(* IEC 61131-3 sources: TIA2AX/tests/test_projects/expected/HW_2200330_V18/ST80_PLC, 6 files *)

(* ---- HwInputs.st ---- *)
TYPE
	HwInputs : STRUCT
		ST80_1_DM260_EB_Box_Acquisition_Status_1 AT %B1205 : ARRAY[0..2] OF BYTE;
		ST80_1_DM260_EB_Box_Results_Status_1 AT %B1208 : BYTE;
		ST80_1_DM260_EB_Box_Soft_Event_Control_1 AT %B1209 : BYTE;
		ST80_1_DM260_EB_Box_Result_Data_64_bytes_1 AT %B1382 : ARRAY[0..71] OF BYTE;
		ST80_1_DM260_PB_Box_Acquisition_Status_1 AT %B1200 : ARRAY[0..2] OF BYTE;
		ST80_1_DM260_PB_Box_Results_Status_1 AT %B1203 : BYTE;
		ST80_1_DM260_PB_Box_Soft_Event_Control_1 AT %B1204 : BYTE;
		ST80_1_DM260_PB_Box_Result_Data_64_bytes_1 AT %B1210 : ARRAY[0..71] OF BYTE;
		ST80_ET200SP_2_11M1 AT %B600 : DWORD;
		ST80_ET200SP_2_11M2 AT %B604 : DWORD;
		ST80_ET200SP_2_11M3 AT %B608 : DWORD;
		ST80_ET200SP_2_11M4 AT %B612 : DWORD;
		ST80_ET200SP_2_12M1 AT %B616 : DWORD;
		ST80_ET200SP_2_12M2 AT %B620 : DWORD;
		ST80_ET200SP_2_12M3 AT %B624 : DWORD;
		ST80_ET200SP_2_12M4 AT %B628 : DWORD;
		ST80_ET200SP_2_13M1 AT %B632 : DWORD;
		ST80_ET200SP_2_13M2 AT %B636 : DWORD;
		ST80_ET200SP_2_13M3 AT %B640 : DWORD;
		ST80_ET200SP_2_13M4 AT %B644 : DWORD;
		ST80_1_TZ535_PN_In_Out_32_byte_1 AT %B1800 : ARRAY[0..31] OF BYTE;
		ST80_1_DM260_Housing_Acquisition_Status_1 AT %B1000 : ARRAY[0..2] OF BYTE;
		ST80_1_DM260_Housing_Results_Status_1 AT %B1003 : BYTE;
		ST80_1_DM260_Housing_Soft_Event_Control_1 AT %B1004 : BYTE;
		ST80_1_DM260_Housing_Result_Data_64_bytes_1 AT %B1010 : ARRAY[0..71] OF BYTE;
		ST80_ET200SP_CM_4xIO_Link_1 AT %B100 : ARRAY[0..31] OF BYTE;
		ST80_ET200SP_CM_4xIO_Link_2 AT %B132 : ARRAY[0..31] OF BYTE;
		ST80_ET200SP_CM_4xIO_Link_3 AT %B164 : ARRAY[0..31] OF BYTE;
		ST80_ET200SP_DI_16x24VDC_ST_1 AT %B0 : WORD;
		ST80_ET200SP_DI_16x24VDC_ST_2 AT %B2 : WORD;
		ST80_ET200SP_DI_16x24VDC_ST_3 AT %B4 : WORD;
		ST80_ET200SP_DI_16x24VDC_ST_4 AT %B6 : WORD;
	END_STRUCT;
END_TYPE

(* ---- HwOutputs.st ---- *)
TYPE
	HwOutputs : STRUCT
		ST80_1_DM260_EB_Box_Acquisition_Control_1 AT %B1201 : BYTE;
		ST80_1_DM260_EB_Box_Results_Control_1 AT %B1205 : BYTE;
		ST80_1_DM260_EB_Box_Soft_Event_Control_1 AT %B1206 : BYTE;
		ST80_1_DM260_EB_Box_User_Data_64_bytes_1 AT %B1378 : ARRAY[0..67] OF BYTE;
		ST80_1_DM260_PB_Box_Acquisition_Control_1 AT %B1200 : BYTE;
		ST80_1_DM260_PB_Box_Results_Control_1 AT %B1203 : BYTE;
		ST80_1_DM260_PB_Box_Soft_Event_Control_1 AT %B1204 : BYTE;
		ST80_1_DM260_PB_Box_User_Data_64_bytes_1 AT %B1210 : ARRAY[0..67] OF BYTE;
		ST80_ET200SP_2_11M1 AT %B600 : WORD;
		ST80_ET200SP_2_11M2 AT %B604 : WORD;
		ST80_ET200SP_2_11M3 AT %B608 : WORD;
		ST80_ET200SP_2_11M4 AT %B612 : WORD;
		ST80_ET200SP_2_12M1 AT %B616 : WORD;
		ST80_ET200SP_2_12M2 AT %B620 : WORD;
		ST80_ET200SP_2_12M3 AT %B624 : WORD;
		ST80_ET200SP_2_12M4 AT %B628 : WORD;
		ST80_ET200SP_2_13M1 AT %B632 : WORD;
		ST80_ET200SP_2_13M2 AT %B636 : WORD;
		ST80_ET200SP_2_13M3 AT %B640 : WORD;
		ST80_ET200SP_2_13M4 AT %B644 : WORD;
		ST80_1_TZ535_PN_In_Out_32_byte_1 AT %B1800 : ARRAY[0..31] OF BYTE;
		ST80_1_DM260_Housing_Acquisition_Control_1 AT %B1000 : BYTE;
		ST80_1_DM260_Housing_Results_Control_1 AT %B1003 : BYTE;
		ST80_1_DM260_Housing_Soft_Event_Control_1 AT %B1004 : BYTE;
		ST80_1_DM260_Housing_User_Data_64_bytes_1 AT %B1010 : ARRAY[0..67] OF BYTE;
		ST80_CPX_MPA1S_VMPA1_FB_EMS_8_8DO_1 AT %B200 : BYTE;
		ST80_CPX_MPA1S_VMPA1_FB_EMS_8_8DO_2 AT %B201 : BYTE;
		ST80_CPX_MPA2S_VMPA2_FB_EMS_4_4DO_1 AT %B202 : BYTE;
		ST80_CPX_MPA1S_VMPA1_FB_EMS_8_8DO_3 AT %B203 : BYTE;
		ST80_CPX_MPA2S_VMPA2_FB_EMS_4_4DO_2 AT %B204 : BYTE;
		ST80_CPX_MPA1S_VMPA1_FB_EMS_8_8DO_4 AT %B205 : BYTE;
		ST80_CPX_MPA1S_VMPA1_FB_EMS_8_8DO_5 AT %B206 : BYTE;
		ST80_CPX_MPA1G_VMPA1_FB_EMG_8_8DO_1 AT %B207 : BYTE;
		ST80_CPX_MPA1G_VMPA1_FB_EMG_8_8DO_2 AT %B208 : BYTE;
		ST80_CPX_MPA2G_VMPA2_FB_EMG_4_4DO_1 AT %B209 : BYTE;
		ST80_CPX_MPA1G_VMPA1_FB_EMG_8_8DO_3 AT %B210 : BYTE;
		ST80_CPX_MPA1G_VMPA1_FB_EMG_8_8DO_4 AT %B211 : BYTE;
		ST80_CPX_MPA1G_VMPA1_FB_EMG_8_8DO_5 AT %B212 : BYTE;
		ST80_CPX_MPA1G_VMPA1_FB_EMG_8_8DO_6 AT %B213 : BYTE;
		ST80_ET200SP_CM_4xIO_Link_1 AT %B100 : ARRAY[0..31] OF BYTE;
		ST80_ET200SP_CM_4xIO_Link_2 AT %B132 : ARRAY[0..31] OF BYTE;
		ST80_ET200SP_CM_4xIO_Link_3 AT %B164 : ARRAY[0..31] OF BYTE;
		ST80_ET200SP_DQ_16x24VDC_0_5A_ST_1 AT %B0 : WORD;
		ST80_ET200SP_DQ_16x24VDC_0_5A_ST_2 AT %B2 : WORD;
		ST80_ET200SP_DQ_16x24VDC_0_5A_ST_3 AT %B4 : WORD;
	END_STRUCT;
END_TYPE

(* ---- PlcInputs.st ---- *)
TYPE
	PlcInputs : STRUCT
		ST80_1_DM260_EB_Box_Acquisition_Status_1 : ARRAY[0..2] OF BYTE;
		ST80_1_DM260_EB_Box_Results_Status_1 : BYTE;
		ST80_1_DM260_EB_Box_Soft_Event_Control_1 : BYTE;
		ST80_1_DM260_EB_Box_Result_Data_64_bytes_1 : ARRAY[0..71] OF BYTE;
		ST80_1_DM260_PB_Box_Acquisition_Status_1 : ARRAY[0..2] OF BYTE;
		ST80_1_DM260_PB_Box_Results_Status_1 : BYTE;
		ST80_1_DM260_PB_Box_Soft_Event_Control_1 : BYTE;
		ST80_1_DM260_PB_Box_Result_Data_64_bytes_1 : ARRAY[0..71] OF BYTE;
		ST80_ET200SP_2_11M1 : DWORD;
		ST80_ET200SP_2_11M2 : DWORD;
		ST80_ET200SP_2_11M3 : DWORD;
		ST80_ET200SP_2_11M4 : DWORD;
		ST80_ET200SP_2_12M1 : DWORD;
		ST80_ET200SP_2_12M2 : DWORD;
		ST80_ET200SP_2_12M3 : DWORD;
		ST80_ET200SP_2_12M4 : DWORD;
		ST80_ET200SP_2_13M1 : DWORD;
		ST80_ET200SP_2_13M2 : DWORD;
		ST80_ET200SP_2_13M3 : DWORD;
		ST80_ET200SP_2_13M4 : DWORD;
		ST80_1_TZ535_PN_In_Out_32_byte_1 : ARRAY[0..31] OF BYTE;
		ST80_1_DM260_Housing_Acquisition_Status_1 : ARRAY[0..2] OF BYTE;
		ST80_1_DM260_Housing_Results_Status_1 : BYTE;
		ST80_1_DM260_Housing_Soft_Event_Control_1 : BYTE;
		ST80_1_DM260_Housing_Result_Data_64_bytes_1 : ARRAY[0..71] OF BYTE;
		ST80_ET200SP_CM_4xIO_Link_1 : ARRAY[0..31] OF BYTE;
		ST80_ET200SP_CM_4xIO_Link_2 : ARRAY[0..31] OF BYTE;
		ST80_ET200SP_CM_4xIO_Link_3 : ARRAY[0..31] OF BYTE;
		ST80_ET200SP_DI_16x24VDC_ST_1 : WORD;
		ST80_ET200SP_DI_16x24VDC_ST_2 : WORD;
		ST80_ET200SP_DI_16x24VDC_ST_3 : WORD;
		ST80_ET200SP_DI_16x24VDC_ST_4 : WORD;
	END_STRUCT;
END_TYPE

(* ---- PlcOutputs.st ---- *)
TYPE
	PlcOutputs : STRUCT
		ST80_1_DM260_EB_Box_Acquisition_Control_1 : BYTE;
		ST80_1_DM260_EB_Box_Results_Control_1 : BYTE;
		ST80_1_DM260_EB_Box_Soft_Event_Control_1 : BYTE;
		ST80_1_DM260_EB_Box_User_Data_64_bytes_1 : ARRAY[0..67] OF BYTE;
		ST80_1_DM260_PB_Box_Acquisition_Control_1 : BYTE;
		ST80_1_DM260_PB_Box_Results_Control_1 : BYTE;
		ST80_1_DM260_PB_Box_Soft_Event_Control_1 : BYTE;
		ST80_1_DM260_PB_Box_User_Data_64_bytes_1 : ARRAY[0..67] OF BYTE;
		ST80_ET200SP_2_11M1 : WORD;
		ST80_ET200SP_2_11M2 : WORD;
		ST80_ET200SP_2_11M3 : WORD;
		ST80_ET200SP_2_11M4 : WORD;
		ST80_ET200SP_2_12M1 : WORD;
		ST80_ET200SP_2_12M2 : WORD;
		ST80_ET200SP_2_12M3 : WORD;
		ST80_ET200SP_2_12M4 : WORD;
		ST80_ET200SP_2_13M1 : WORD;
		ST80_ET200SP_2_13M2 : WORD;
		ST80_ET200SP_2_13M3 : WORD;
		ST80_ET200SP_2_13M4 : WORD;
		ST80_1_TZ535_PN_In_Out_32_byte_1 : ARRAY[0..31] OF BYTE;
		ST80_1_DM260_Housing_Acquisition_Control_1 : BYTE;
		ST80_1_DM260_Housing_Results_Control_1 : BYTE;
		ST80_1_DM260_Housing_Soft_Event_Control_1 : BYTE;
		ST80_1_DM260_Housing_User_Data_64_bytes_1 : ARRAY[0..67] OF BYTE;
		ST80_CPX_MPA1S_VMPA1_FB_EMS_8_8DO_1 : BYTE;
		ST80_CPX_MPA1S_VMPA1_FB_EMS_8_8DO_2 : BYTE;
		ST80_CPX_MPA2S_VMPA2_FB_EMS_4_4DO_1 : BYTE;
		ST80_CPX_MPA1S_VMPA1_FB_EMS_8_8DO_3 : BYTE;
		ST80_CPX_MPA2S_VMPA2_FB_EMS_4_4DO_2 : BYTE;
		ST80_CPX_MPA1S_VMPA1_FB_EMS_8_8DO_4 : BYTE;
		ST80_CPX_MPA1S_VMPA1_FB_EMS_8_8DO_5 : BYTE;
		ST80_CPX_MPA1G_VMPA1_FB_EMG_8_8DO_1 : BYTE;
		ST80_CPX_MPA1G_VMPA1_FB_EMG_8_8DO_2 : BYTE;
		ST80_CPX_MPA2G_VMPA2_FB_EMG_4_4DO_1 : BYTE;
		ST80_CPX_MPA1G_VMPA1_FB_EMG_8_8DO_3 : BYTE;
		ST80_CPX_MPA1G_VMPA1_FB_EMG_8_8DO_4 : BYTE;
		ST80_CPX_MPA1G_VMPA1_FB_EMG_8_8DO_5 : BYTE;
		ST80_CPX_MPA1G_VMPA1_FB_EMG_8_8DO_6 : BYTE;
		ST80_ET200SP_CM_4xIO_Link_1 : ARRAY[0..31] OF BYTE;
		ST80_ET200SP_CM_4xIO_Link_2 : ARRAY[0..31] OF BYTE;
		ST80_ET200SP_CM_4xIO_Link_3 : ARRAY[0..31] OF BYTE;
		ST80_ET200SP_DQ_16x24VDC_0_5A_ST_1 : WORD;
		ST80_ET200SP_DQ_16x24VDC_0_5A_ST_2 : WORD;
		ST80_ET200SP_DQ_16x24VDC_0_5A_ST_3 : WORD;
	END_STRUCT;
END_TYPE

(* ---- CopyInputs.st ---- *)
FUNCTION CopyInputs
	VAR_EXTERNAL
		HwInputs : HwInputs;
		PlcInputs : PlcInputs;
	END_VAR
	PlcInputs.ST80_1_DM260_EB_Box_Acquisition_Status_1[0] := HwInputs.ST80_1_DM260_EB_Box_Acquisition_Status_1[0];
	PlcInputs.ST80_1_DM260_EB_Box_Acquisition_Status_1[1] := HwInputs.ST80_1_DM260_EB_Box_Acquisition_Status_1[1];
	PlcInputs.ST80_1_DM260_EB_Box_Acquisition_Status_1[2] := HwInputs.ST80_1_DM260_EB_Box_Acquisition_Status_1[2];
	PlcInputs.ST80_1_DM260_EB_Box_Results_Status_1 := HwInputs.ST80_1_DM260_EB_Box_Results_Status_1;
	PlcInputs.ST80_1_DM260_EB_Box_Soft_Event_Control_1 := HwInputs.ST80_1_DM260_EB_Box_Soft_Event_Control_1;
	PlcInputs.ST80_1_DM260_EB_Box_Result_Data_64_bytes_1[0] := HwInputs.ST80_1_DM260_EB_Box_Result_Data_64_bytes_1[0];
	PlcInputs.ST80_1_DM260_EB_Box_Result_Data_64_bytes_1[1] := HwInputs.ST80_1_DM260_EB_Box_Result_Data_64_bytes_1[1];
	PlcInputs.ST80_1_DM260_EB_Box_Result_Data_64_bytes_1[2] := HwInputs.ST80_1_DM260_EB_Box_Result_Data_64_bytes_1[2];
	PlcInputs.ST80_1_DM260_EB_Box_Result_Data_64_bytes_1[3] := HwInputs.ST80_1_DM260_EB_Box_Result_Data_64_bytes_1[3];
	PlcInputs.ST80_1_DM260_EB_Box_Result_Data_64_bytes_1[4] := HwInputs.ST80_1_DM260_EB_Box_Result_Data_64_bytes_1[4];
	PlcInputs.ST80_1_DM260_EB_Box_Result_Data_64_bytes_1[5] := HwInputs.ST80_1_DM260_EB_Box_Result_Data_64_bytes_1[5];
	PlcInputs.ST80_1_DM260_EB_Box_Result_Data_64_bytes_1[6] := HwInputs.ST80_1_DM260_EB_Box_Result_Data_64_bytes_1[6];
	PlcInputs.ST80_1_DM260_EB_Box_Result_Data_64_bytes_1[7] := HwInputs.ST80_1_DM260_EB_Box_Result_Data_64_bytes_1[7];
	PlcInputs.ST80_1_DM260_EB_Box_Result_Data_64_bytes_1[8] := HwInputs.ST80_1_DM260_EB_Box_Result_Data_64_bytes_1[8];
	PlcInputs.ST80_1_DM260_EB_Box_Result_Data_64_bytes_1[9] := HwInputs.ST80_1_DM260_EB_Box_Result_Data_64_bytes_1[9];
	PlcInputs.ST80_1_DM260_EB_Box_Result_Data_64_bytes_1[10] := HwInputs.ST80_1_DM260_EB_Box_Result_Data_64_bytes_1[10];
	PlcInputs.ST80_1_DM260_EB_Box_Result_Data_64_bytes_1[11] := HwInputs.ST80_1_DM260_EB_Box_Result_Data_64_bytes_1[11];
	PlcInputs.ST80_1_DM260_EB_Box_Result_Data_64_bytes_1[12] := HwInputs.ST80_1_DM260_EB_Box_Result_Data_64_bytes_1[12];
	PlcInputs.ST80_1_DM260_EB_Box_Result_Data_64_bytes_1[13] := HwInputs.ST80_1_DM260_EB_Box_Result_Data_64_bytes_1[13];
	PlcInputs.ST80_1_DM260_EB_Box_Result_Data_64_bytes_1[14] := HwInputs.ST80_1_DM260_EB_Box_Result_Data_64_bytes_1[14];
	PlcInputs.ST80_1_DM260_EB_Box_Result_Data_64_bytes_1[15] := HwInputs.ST80_1_DM260_EB_Box_Result_Data_64_bytes_1[15];
	PlcInputs.ST80_1_DM260_EB_Box_Result_Data_64_bytes_1[16] := HwInputs.ST80_1_DM260_EB_Box_Result_Data_64_bytes_1[16];
	PlcInputs.ST80_1_DM260_EB_Box_Result_Data_64_bytes_1[17] := HwInputs.ST80_1_DM260_EB_Box_Result_Data_64_bytes_1[17];
	PlcInputs.ST80_1_DM260_EB_Box_Result_Data_64_bytes_1[18] := HwInputs.ST80_1_DM260_EB_Box_Result_Data_64_bytes_1[18];
	PlcInputs.ST80_1_DM260_EB_Box_Result_Data_64_bytes_1[19] := HwInputs.ST80_1_DM260_EB_Box_Result_Data_64_bytes_1[19];
	PlcInputs.ST80_1_DM260_EB_Box_Result_Data_64_bytes_1[20] := HwInputs.ST80_1_DM260_EB_Box_Result_Data_64_bytes_1[20];
	PlcInputs.ST80_1_DM260_EB_Box_Result_Data_64_bytes_1[21] := HwInputs.ST80_1_DM260_EB_Box_Result_Data_64_bytes_1[21];
	PlcInputs.ST80_1_DM260_EB_Box_Result_Data_64_bytes_1[22] := HwInputs.ST80_1_DM260_EB_Box_Result_Data_64_bytes_1[22];
	PlcInputs.ST80_1_DM260_EB_Box_Result_Data_64_bytes_1[23] := HwInputs.ST80_1_DM260_EB_Box_Result_Data_64_bytes_1[23];
	PlcInputs.ST80_1_DM260_EB_Box_Result_Data_64_bytes_1[24] := HwInputs.ST80_1_DM260_EB_Box_Result_Data_64_bytes_1[24];
	PlcInputs.ST80_1_DM260_EB_Box_Result_Data_64_bytes_1[25] := HwInputs.ST80_1_DM260_EB_Box_Result_Data_64_bytes_1[25];
	PlcInputs.ST80_1_DM260_EB_Box_Result_Data_64_bytes_1[26] := HwInputs.ST80_1_DM260_EB_Box_Result_Data_64_bytes_1[26];
	PlcInputs.ST80_1_DM260_EB_Box_Result_Data_64_bytes_1[27] := HwInputs.ST80_1_DM260_EB_Box_Result_Data_64_bytes_1[27];
	PlcInputs.ST80_1_DM260_EB_Box_Result_Data_64_bytes_1[28] := HwInputs.ST80_1_DM260_EB_Box_Result_Data_64_bytes_1[28];
	PlcInputs.ST80_1_DM260_EB_Box_Result_Data_64_bytes_1[29] := HwInputs.ST80_1_DM260_EB_Box_Result_Data_64_bytes_1[29];
	PlcInputs.ST80_1_DM260_EB_Box_Result_Data_64_bytes_1[30] := HwInputs.ST80_1_DM260_EB_Box_Result_Data_64_bytes_1[30];
	PlcInputs.ST80_1_DM260_EB_Box_Result_Data_64_bytes_1[31] := HwInputs.ST80_1_DM260_EB_Box_Result_Data_64_bytes_1[31];
	PlcInputs.ST80_1_DM260_EB_Box_Result_Data_64_bytes_1[32] := HwInputs.ST80_1_DM260_EB_Box_Result_Data_64_bytes_1[32];
	PlcInputs.ST80_1_DM260_EB_Box_Result_Data_64_bytes_1[33] := HwInputs.ST80_1_DM260_EB_Box_Result_Data_64_bytes_1[33];
	PlcInputs.ST80_1_DM260_EB_Box_Result_Data_64_bytes_1[34] := HwInputs.ST80_1_DM260_EB_Box_Result_Data_64_bytes_1[34];
	PlcInputs.ST80_1_DM260_EB_Box_Result_Data_64_bytes_1[35] := HwInputs.ST80_1_DM260_EB_Box_Result_Data_64_bytes_1[35];
	PlcInputs.ST80_1_DM260_EB_Box_Result_Data_64_bytes_1[36] := HwInputs.ST80_1_DM260_EB_Box_Result_Data_64_bytes_1[36];
	PlcInputs.ST80_1_DM260_EB_Box_Result_Data_64_bytes_1[37] := HwInputs.ST80_1_DM260_EB_Box_Result_Data_64_bytes_1[37];
	PlcInputs.ST80_1_DM260_EB_Box_Result_Data_64_bytes_1[38] := HwInputs.ST80_1_DM260_EB_Box_Result_Data_64_bytes_1[38];
	PlcInputs.ST80_1_DM260_EB_Box_Result_Data_64_bytes_1[39] := HwInputs.ST80_1_DM260_EB_Box_Result_Data_64_bytes_1[39];
	PlcInputs.ST80_1_DM260_EB_Box_Result_Data_64_bytes_1[40] := HwInputs.ST80_1_DM260_EB_Box_Result_Data_64_bytes_1[40];
	PlcInputs.ST80_1_DM260_EB_Box_Result_Data_64_bytes_1[41] := HwInputs.ST80_1_DM260_EB_Box_Result_Data_64_bytes_1[41];
	PlcInputs.ST80_1_DM260_EB_Box_Result_Data_64_bytes_1[42] := HwInputs.ST80_1_DM260_EB_Box_Result_Data_64_bytes_1[42];
	PlcInputs.ST80_1_DM260_EB_Box_Result_Data_64_bytes_1[43] := HwInputs.ST80_1_DM260_EB_Box_Result_Data_64_bytes_1[43];
	PlcInputs.ST80_1_DM260_EB_Box_Result_Data_64_bytes_1[44] := HwInputs.ST80_1_DM260_EB_Box_Result_Data_64_bytes_1[44];
	PlcInputs.ST80_1_DM260_EB_Box_Result_Data_64_bytes_1[45] := HwInputs.ST80_1_DM260_EB_Box_Result_Data_64_bytes_1[45];
	PlcInputs.ST80_1_DM260_EB_Box_Result_Data_64_bytes_1[46] := HwInputs.ST80_1_DM260_EB_Box_Result_Data_64_bytes_1[46];
	PlcInputs.ST80_1_DM260_EB_Box_Result_Data_64_bytes_1[47] := HwInputs.ST80_1_DM260_EB_Box_Result_Data_64_bytes_1[47];
	PlcInputs.ST80_1_DM260_EB_Box_Result_Data_64_bytes_1[48] := HwInputs.ST80_1_DM260_EB_Box_Result_Data_64_bytes_1[48];
	PlcInputs.ST80_1_DM260_EB_Box_Result_Data_64_bytes_1[49] := HwInputs.ST80_1_DM260_EB_Box_Result_Data_64_bytes_1[49];
	PlcInputs.ST80_1_DM260_EB_Box_Result_Data_64_bytes_1[50] := HwInputs.ST80_1_DM260_EB_Box_Result_Data_64_bytes_1[50];
	PlcInputs.ST80_1_DM260_EB_Box_Result_Data_64_bytes_1[51] := HwInputs.ST80_1_DM260_EB_Box_Result_Data_64_bytes_1[51];
	PlcInputs.ST80_1_DM260_EB_Box_Result_Data_64_bytes_1[52] := HwInputs.ST80_1_DM260_EB_Box_Result_Data_64_bytes_1[52];
	PlcInputs.ST80_1_DM260_EB_Box_Result_Data_64_bytes_1[53] := HwInputs.ST80_1_DM260_EB_Box_Result_Data_64_bytes_1[53];
	PlcInputs.ST80_1_DM260_EB_Box_Result_Data_64_bytes_1[54] := HwInputs.ST80_1_DM260_EB_Box_Result_Data_64_bytes_1[54];
	PlcInputs.ST80_1_DM260_EB_Box_Result_Data_64_bytes_1[55] := HwInputs.ST80_1_DM260_EB_Box_Result_Data_64_bytes_1[55];
	PlcInputs.ST80_1_DM260_EB_Box_Result_Data_64_bytes_1[56] := HwInputs.ST80_1_DM260_EB_Box_Result_Data_64_bytes_1[56];
	PlcInputs.ST80_1_DM260_EB_Box_Result_Data_64_bytes_1[57] := HwInputs.ST80_1_DM260_EB_Box_Result_Data_64_bytes_1[57];
	PlcInputs.ST80_1_DM260_EB_Box_Result_Data_64_bytes_1[58] := HwInputs.ST80_1_DM260_EB_Box_Result_Data_64_bytes_1[58];
	PlcInputs.ST80_1_DM260_EB_Box_Result_Data_64_bytes_1[59] := HwInputs.ST80_1_DM260_EB_Box_Result_Data_64_bytes_1[59];
	PlcInputs.ST80_1_DM260_EB_Box_Result_Data_64_bytes_1[60] := HwInputs.ST80_1_DM260_EB_Box_Result_Data_64_bytes_1[60];
	PlcInputs.ST80_1_DM260_EB_Box_Result_Data_64_bytes_1[61] := HwInputs.ST80_1_DM260_EB_Box_Result_Data_64_bytes_1[61];
	PlcInputs.ST80_1_DM260_EB_Box_Result_Data_64_bytes_1[62] := HwInputs.ST80_1_DM260_EB_Box_Result_Data_64_bytes_1[62];
	PlcInputs.ST80_1_DM260_EB_Box_Result_Data_64_bytes_1[63] := HwInputs.ST80_1_DM260_EB_Box_Result_Data_64_bytes_1[63];
	PlcInputs.ST80_1_DM260_EB_Box_Result_Data_64_bytes_1[64] := HwInputs.ST80_1_DM260_EB_Box_Result_Data_64_bytes_1[64];
	PlcInputs.ST80_1_DM260_EB_Box_Result_Data_64_bytes_1[65] := HwInputs.ST80_1_DM260_EB_Box_Result_Data_64_bytes_1[65];
	PlcInputs.ST80_1_DM260_EB_Box_Result_Data_64_bytes_1[66] := HwInputs.ST80_1_DM260_EB_Box_Result_Data_64_bytes_1[66];
	PlcInputs.ST80_1_DM260_EB_Box_Result_Data_64_bytes_1[67] := HwInputs.ST80_1_DM260_EB_Box_Result_Data_64_bytes_1[67];
	PlcInputs.ST80_1_DM260_EB_Box_Result_Data_64_bytes_1[68] := HwInputs.ST80_1_DM260_EB_Box_Result_Data_64_bytes_1[68];
	PlcInputs.ST80_1_DM260_EB_Box_Result_Data_64_bytes_1[69] := HwInputs.ST80_1_DM260_EB_Box_Result_Data_64_bytes_1[69];
	PlcInputs.ST80_1_DM260_EB_Box_Result_Data_64_bytes_1[70] := HwInputs.ST80_1_DM260_EB_Box_Result_Data_64_bytes_1[70];
	PlcInputs.ST80_1_DM260_EB_Box_Result_Data_64_bytes_1[71] := HwInputs.ST80_1_DM260_EB_Box_Result_Data_64_bytes_1[71];
	PlcInputs.ST80_1_DM260_PB_Box_Acquisition_Status_1[0] := HwInputs.ST80_1_DM260_PB_Box_Acquisition_Status_1[0];
	PlcInputs.ST80_1_DM260_PB_Box_Acquisition_Status_1[1] := HwInputs.ST80_1_DM260_PB_Box_Acquisition_Status_1[1];
	PlcInputs.ST80_1_DM260_PB_Box_Acquisition_Status_1[2] := HwInputs.ST80_1_DM260_PB_Box_Acquisition_Status_1[2];
	PlcInputs.ST80_1_DM260_PB_Box_Results_Status_1 := HwInputs.ST80_1_DM260_PB_Box_Results_Status_1;
	PlcInputs.ST80_1_DM260_PB_Box_Soft_Event_Control_1 := HwInputs.ST80_1_DM260_PB_Box_Soft_Event_Control_1;
	PlcInputs.ST80_1_DM260_PB_Box_Result_Data_64_bytes_1[0] := HwInputs.ST80_1_DM260_PB_Box_Result_Data_64_bytes_1[0];
	PlcInputs.ST80_1_DM260_PB_Box_Result_Data_64_bytes_1[1] := HwInputs.ST80_1_DM260_PB_Box_Result_Data_64_bytes_1[1];
	PlcInputs.ST80_1_DM260_PB_Box_Result_Data_64_bytes_1[2] := HwInputs.ST80_1_DM260_PB_Box_Result_Data_64_bytes_1[2];
	PlcInputs.ST80_1_DM260_PB_Box_Result_Data_64_bytes_1[3] := HwInputs.ST80_1_DM260_PB_Box_Result_Data_64_bytes_1[3];
	PlcInputs.ST80_1_DM260_PB_Box_Result_Data_64_bytes_1[4] := HwInputs.ST80_1_DM260_PB_Box_Result_Data_64_bytes_1[4];
	PlcInputs.ST80_1_DM260_PB_Box_Result_Data_64_bytes_1[5] := HwInputs.ST80_1_DM260_PB_Box_Result_Data_64_bytes_1[5];
	PlcInputs.ST80_1_DM260_PB_Box_Result_Data_64_bytes_1[6] := HwInputs.ST80_1_DM260_PB_Box_Result_Data_64_bytes_1[6];
	PlcInputs.ST80_1_DM260_PB_Box_Result_Data_64_bytes_1[7] := HwInputs.ST80_1_DM260_PB_Box_Result_Data_64_bytes_1[7];
	PlcInputs.ST80_1_DM260_PB_Box_Result_Data_64_bytes_1[8] := HwInputs.ST80_1_DM260_PB_Box_Result_Data_64_bytes_1[8];
	PlcInputs.ST80_1_DM260_PB_Box_Result_Data_64_bytes_1[9] := HwInputs.ST80_1_DM260_PB_Box_Result_Data_64_bytes_1[9];
	PlcInputs.ST80_1_DM260_PB_Box_Result_Data_64_bytes_1[10] := HwInputs.ST80_1_DM260_PB_Box_Result_Data_64_bytes_1[10];
	PlcInputs.ST80_1_DM260_PB_Box_Result_Data_64_bytes_1[11] := HwInputs.ST80_1_DM260_PB_Box_Result_Data_64_bytes_1[11];
	PlcInputs.ST80_1_DM260_PB_Box_Result_Data_64_bytes_1[12] := HwInputs.ST80_1_DM260_PB_Box_Result_Data_64_bytes_1[12];
	PlcInputs.ST80_1_DM260_PB_Box_Result_Data_64_bytes_1[13] := HwInputs.ST80_1_DM260_PB_Box_Result_Data_64_bytes_1[13];
	PlcInputs.ST80_1_DM260_PB_Box_Result_Data_64_bytes_1[14] := HwInputs.ST80_1_DM260_PB_Box_Result_Data_64_bytes_1[14];
	PlcInputs.ST80_1_DM260_PB_Box_Result_Data_64_bytes_1[15] := HwInputs.ST80_1_DM260_PB_Box_Result_Data_64_bytes_1[15];
	PlcInputs.ST80_1_DM260_PB_Box_Result_Data_64_bytes_1[16] := HwInputs.ST80_1_DM260_PB_Box_Result_Data_64_bytes_1[16];
	PlcInputs.ST80_1_DM260_PB_Box_Result_Data_64_bytes_1[17] := HwInputs.ST80_1_DM260_PB_Box_Result_Data_64_bytes_1[17];
	PlcInputs.ST80_1_DM260_PB_Box_Result_Data_64_bytes_1[18] := HwInputs.ST80_1_DM260_PB_Box_Result_Data_64_bytes_1[18];
	PlcInputs.ST80_1_DM260_PB_Box_Result_Data_64_bytes_1[19] := HwInputs.ST80_1_DM260_PB_Box_Result_Data_64_bytes_1[19];
	PlcInputs.ST80_1_DM260_PB_Box_Result_Data_64_bytes_1[20] := HwInputs.ST80_1_DM260_PB_Box_Result_Data_64_bytes_1[20];
	PlcInputs.ST80_1_DM260_PB_Box_Result_Data_64_bytes_1[21] := HwInputs.ST80_1_DM260_PB_Box_Result_Data_64_bytes_1[21];
	PlcInputs.ST80_1_DM260_PB_Box_Result_Data_64_bytes_1[22] := HwInputs.ST80_1_DM260_PB_Box_Result_Data_64_bytes_1[22];
	PlcInputs.ST80_1_DM260_PB_Box_Result_Data_64_bytes_1[23] := HwInputs.ST80_1_DM260_PB_Box_Result_Data_64_bytes_1[23];
	PlcInputs.ST80_1_DM260_PB_Box_Result_Data_64_bytes_1[24] := HwInputs.ST80_1_DM260_PB_Box_Result_Data_64_bytes_1[24];
	PlcInputs.ST80_1_DM260_PB_Box_Result_Data_64_bytes_1[25] := HwInputs.ST80_1_DM260_PB_Box_Result_Data_64_bytes_1[25];
	PlcInputs.ST80_1_DM260_PB_Box_Result_Data_64_bytes_1[26] := HwInputs.ST80_1_DM260_PB_Box_Result_Data_64_bytes_1[26];
	PlcInputs.ST80_1_DM260_PB_Box_Result_Data_64_bytes_1[27] := HwInputs.ST80_1_DM260_PB_Box_Result_Data_64_bytes_1[27];
	PlcInputs.ST80_1_DM260_PB_Box_Result_Data_64_bytes_1[28] := HwInputs.ST80_1_DM260_PB_Box_Result_Data_64_bytes_1[28];
	PlcInputs.ST80_1_DM260_PB_Box_Result_Data_64_bytes_1[29] := HwInputs.ST80_1_DM260_PB_Box_Result_Data_64_bytes_1[29];
	PlcInputs.ST80_1_DM260_PB_Box_Result_Data_64_bytes_1[30] := HwInputs.ST80_1_DM260_PB_Box_Result_Data_64_bytes_1[30];
	PlcInputs.ST80_1_DM260_PB_Box_Result_Data_64_bytes_1[31] := HwInputs.ST80_1_DM260_PB_Box_Result_Data_64_bytes_1[31];
	PlcInputs.ST80_1_DM260_PB_Box_Result_Data_64_bytes_1[32] := HwInputs.ST80_1_DM260_PB_Box_Result_Data_64_bytes_1[32];
	PlcInputs.ST80_1_DM260_PB_Box_Result_Data_64_bytes_1[33] := HwInputs.ST80_1_DM260_PB_Box_Result_Data_64_bytes_1[33];
	PlcInputs.ST80_1_DM260_PB_Box_Result_Data_64_bytes_1[34] := HwInputs.ST80_1_DM260_PB_Box_Result_Data_64_bytes_1[34];
	PlcInputs.ST80_1_DM260_PB_Box_Result_Data_64_bytes_1[35] := HwInputs.ST80_1_DM260_PB_Box_Result_Data_64_bytes_1[35];
	PlcInputs.ST80_1_DM260_PB_Box_Result_Data_64_bytes_1[36] := HwInputs.ST80_1_DM260_PB_Box_Result_Data_64_bytes_1[36];
	PlcInputs.ST80_1_DM260_PB_Box_Result_Data_64_bytes_1[37] := HwInputs.ST80_1_DM260_PB_Box_Result_Data_64_bytes_1[37];
	PlcInputs.ST80_1_DM260_PB_Box_Result_Data_64_bytes_1[38] := HwInputs.ST80_1_DM260_PB_Box_Result_Data_64_bytes_1[38];
	PlcInputs.ST80_1_DM260_PB_Box_Result_Data_64_bytes_1[39] := HwInputs.ST80_1_DM260_PB_Box_Result_Data_64_bytes_1[39];
	PlcInputs.ST80_1_DM260_PB_Box_Result_Data_64_bytes_1[40] := HwInputs.ST80_1_DM260_PB_Box_Result_Data_64_bytes_1[40];
	PlcInputs.ST80_1_DM260_PB_Box_Result_Data_64_bytes_1[41] := HwInputs.ST80_1_DM260_PB_Box_Result_Data_64_bytes_1[41];
	PlcInputs.ST80_1_DM260_PB_Box_Result_Data_64_bytes_1[42] := HwInputs.ST80_1_DM260_PB_Box_Result_Data_64_bytes_1[42];
	PlcInputs.ST80_1_DM260_PB_Box_Result_Data_64_bytes_1[43] := HwInputs.ST80_1_DM260_PB_Box_Result_Data_64_bytes_1[43];
	PlcInputs.ST80_1_DM260_PB_Box_Result_Data_64_bytes_1[44] := HwInputs.ST80_1_DM260_PB_Box_Result_Data_64_bytes_1[44];
	PlcInputs.ST80_1_DM260_PB_Box_Result_Data_64_bytes_1[45] := HwInputs.ST80_1_DM260_PB_Box_Result_Data_64_bytes_1[45];
	PlcInputs.ST80_1_DM260_PB_Box_Result_Data_64_bytes_1[46] := HwInputs.ST80_1_DM260_PB_Box_Result_Data_64_bytes_1[46];
	PlcInputs.ST80_1_DM260_PB_Box_Result_Data_64_bytes_1[47] := HwInputs.ST80_1_DM260_PB_Box_Result_Data_64_bytes_1[47];
	PlcInputs.ST80_1_DM260_PB_Box_Result_Data_64_bytes_1[48] := HwInputs.ST80_1_DM260_PB_Box_Result_Data_64_bytes_1[48];
	PlcInputs.ST80_1_DM260_PB_Box_Result_Data_64_bytes_1[49] := HwInputs.ST80_1_DM260_PB_Box_Result_Data_64_bytes_1[49];
	PlcInputs.ST80_1_DM260_PB_Box_Result_Data_64_bytes_1[50] := HwInputs.ST80_1_DM260_PB_Box_Result_Data_64_bytes_1[50];
	PlcInputs.ST80_1_DM260_PB_Box_Result_Data_64_bytes_1[51] := HwInputs.ST80_1_DM260_PB_Box_Result_Data_64_bytes_1[51];
	PlcInputs.ST80_1_DM260_PB_Box_Result_Data_64_bytes_1[52] := HwInputs.ST80_1_DM260_PB_Box_Result_Data_64_bytes_1[52];
	PlcInputs.ST80_1_DM260_PB_Box_Result_Data_64_bytes_1[53] := HwInputs.ST80_1_DM260_PB_Box_Result_Data_64_bytes_1[53];
	PlcInputs.ST80_1_DM260_PB_Box_Result_Data_64_bytes_1[54] := HwInputs.ST80_1_DM260_PB_Box_Result_Data_64_bytes_1[54];
	PlcInputs.ST80_1_DM260_PB_Box_Result_Data_64_bytes_1[55] := HwInputs.ST80_1_DM260_PB_Box_Result_Data_64_bytes_1[55];
	PlcInputs.ST80_1_DM260_PB_Box_Result_Data_64_bytes_1[56] := HwInputs.ST80_1_DM260_PB_Box_Result_Data_64_bytes_1[56];
	PlcInputs.ST80_1_DM260_PB_Box_Result_Data_64_bytes_1[57] := HwInputs.ST80_1_DM260_PB_Box_Result_Data_64_bytes_1[57];
	PlcInputs.ST80_1_DM260_PB_Box_Result_Data_64_bytes_1[58] := HwInputs.ST80_1_DM260_PB_Box_Result_Data_64_bytes_1[58];
	PlcInputs.ST80_1_DM260_PB_Box_Result_Data_64_bytes_1[59] := HwInputs.ST80_1_DM260_PB_Box_Result_Data_64_bytes_1[59];
	PlcInputs.ST80_1_DM260_PB_Box_Result_Data_64_bytes_1[60] := HwInputs.ST80_1_DM260_PB_Box_Result_Data_64_bytes_1[60];
	PlcInputs.ST80_1_DM260_PB_Box_Result_Data_64_bytes_1[61] := HwInputs.ST80_1_DM260_PB_Box_Result_Data_64_bytes_1[61];
	PlcInputs.ST80_1_DM260_PB_Box_Result_Data_64_bytes_1[62] := HwInputs.ST80_1_DM260_PB_Box_Result_Data_64_bytes_1[62];
	PlcInputs.ST80_1_DM260_PB_Box_Result_Data_64_bytes_1[63] := HwInputs.ST80_1_DM260_PB_Box_Result_Data_64_bytes_1[63];
	PlcInputs.ST80_1_DM260_PB_Box_Result_Data_64_bytes_1[64] := HwInputs.ST80_1_DM260_PB_Box_Result_Data_64_bytes_1[64];
	PlcInputs.ST80_1_DM260_PB_Box_Result_Data_64_bytes_1[65] := HwInputs.ST80_1_DM260_PB_Box_Result_Data_64_bytes_1[65];
	PlcInputs.ST80_1_DM260_PB_Box_Result_Data_64_bytes_1[66] := HwInputs.ST80_1_DM260_PB_Box_Result_Data_64_bytes_1[66];
	PlcInputs.ST80_1_DM260_PB_Box_Result_Data_64_bytes_1[67] := HwInputs.ST80_1_DM260_PB_Box_Result_Data_64_bytes_1[67];
	PlcInputs.ST80_1_DM260_PB_Box_Result_Data_64_bytes_1[68] := HwInputs.ST80_1_DM260_PB_Box_Result_Data_64_bytes_1[68];
	PlcInputs.ST80_1_DM260_PB_Box_Result_Data_64_bytes_1[69] := HwInputs.ST80_1_DM260_PB_Box_Result_Data_64_bytes_1[69];
	PlcInputs.ST80_1_DM260_PB_Box_Result_Data_64_bytes_1[70] := HwInputs.ST80_1_DM260_PB_Box_Result_Data_64_bytes_1[70];
	PlcInputs.ST80_1_DM260_PB_Box_Result_Data_64_bytes_1[71] := HwInputs.ST80_1_DM260_PB_Box_Result_Data_64_bytes_1[71];
	PlcInputs.ST80_ET200SP_2_11M1 := HwInputs.ST80_ET200SP_2_11M1;
	PlcInputs.ST80_ET200SP_2_11M2 := HwInputs.ST80_ET200SP_2_11M2;
	PlcInputs.ST80_ET200SP_2_11M3 := HwInputs.ST80_ET200SP_2_11M3;
	PlcInputs.ST80_ET200SP_2_11M4 := HwInputs.ST80_ET200SP_2_11M4;
	PlcInputs.ST80_ET200SP_2_12M1 := HwInputs.ST80_ET200SP_2_12M1;
	PlcInputs.ST80_ET200SP_2_12M2 := HwInputs.ST80_ET200SP_2_12M2;
	PlcInputs.ST80_ET200SP_2_12M3 := HwInputs.ST80_ET200SP_2_12M3;
	PlcInputs.ST80_ET200SP_2_12M4 := HwInputs.ST80_ET200SP_2_12M4;
	PlcInputs.ST80_ET200SP_2_13M1 := HwInputs.ST80_ET200SP_2_13M1;
	PlcInputs.ST80_ET200SP_2_13M2 := HwInputs.ST80_ET200SP_2_13M2;
	PlcInputs.ST80_ET200SP_2_13M3 := HwInputs.ST80_ET200SP_2_13M3;
	PlcInputs.ST80_ET200SP_2_13M4 := HwInputs.ST80_ET200SP_2_13M4;
	PlcInputs.ST80_1_TZ535_PN_In_Out_32_byte_1[0] := HwInputs.ST80_1_TZ535_PN_In_Out_32_byte_1[0];
	PlcInputs.ST80_1_TZ535_PN_In_Out_32_byte_1[1] := HwInputs.ST80_1_TZ535_PN_In_Out_32_byte_1[1];
	PlcInputs.ST80_1_TZ535_PN_In_Out_32_byte_1[2] := HwInputs.ST80_1_TZ535_PN_In_Out_32_byte_1[2];
	PlcInputs.ST80_1_TZ535_PN_In_Out_32_byte_1[3] := HwInputs.ST80_1_TZ535_PN_In_Out_32_byte_1[3];
	PlcInputs.ST80_1_TZ535_PN_In_Out_32_byte_1[4] := HwInputs.ST80_1_TZ535_PN_In_Out_32_byte_1[4];
	PlcInputs.ST80_1_TZ535_PN_In_Out_32_byte_1[5] := HwInputs.ST80_1_TZ535_PN_In_Out_32_byte_1[5];
	PlcInputs.ST80_1_TZ535_PN_In_Out_32_byte_1[6] := HwInputs.ST80_1_TZ535_PN_In_Out_32_byte_1[6];
	PlcInputs.ST80_1_TZ535_PN_In_Out_32_byte_1[7] := HwInputs.ST80_1_TZ535_PN_In_Out_32_byte_1[7];
	PlcInputs.ST80_1_TZ535_PN_In_Out_32_byte_1[8] := HwInputs.ST80_1_TZ535_PN_In_Out_32_byte_1[8];
	PlcInputs.ST80_1_TZ535_PN_In_Out_32_byte_1[9] := HwInputs.ST80_1_TZ535_PN_In_Out_32_byte_1[9];
	PlcInputs.ST80_1_TZ535_PN_In_Out_32_byte_1[10] := HwInputs.ST80_1_TZ535_PN_In_Out_32_byte_1[10];
	PlcInputs.ST80_1_TZ535_PN_In_Out_32_byte_1[11] := HwInputs.ST80_1_TZ535_PN_In_Out_32_byte_1[11];
	PlcInputs.ST80_1_TZ535_PN_In_Out_32_byte_1[12] := HwInputs.ST80_1_TZ535_PN_In_Out_32_byte_1[12];
	PlcInputs.ST80_1_TZ535_PN_In_Out_32_byte_1[13] := HwInputs.ST80_1_TZ535_PN_In_Out_32_byte_1[13];
	PlcInputs.ST80_1_TZ535_PN_In_Out_32_byte_1[14] := HwInputs.ST80_1_TZ535_PN_In_Out_32_byte_1[14];
	PlcInputs.ST80_1_TZ535_PN_In_Out_32_byte_1[15] := HwInputs.ST80_1_TZ535_PN_In_Out_32_byte_1[15];
	PlcInputs.ST80_1_TZ535_PN_In_Out_32_byte_1[16] := HwInputs.ST80_1_TZ535_PN_In_Out_32_byte_1[16];
	PlcInputs.ST80_1_TZ535_PN_In_Out_32_byte_1[17] := HwInputs.ST80_1_TZ535_PN_In_Out_32_byte_1[17];
	PlcInputs.ST80_1_TZ535_PN_In_Out_32_byte_1[18] := HwInputs.ST80_1_TZ535_PN_In_Out_32_byte_1[18];
	PlcInputs.ST80_1_TZ535_PN_In_Out_32_byte_1[19] := HwInputs.ST80_1_TZ535_PN_In_Out_32_byte_1[19];
	PlcInputs.ST80_1_TZ535_PN_In_Out_32_byte_1[20] := HwInputs.ST80_1_TZ535_PN_In_Out_32_byte_1[20];
	PlcInputs.ST80_1_TZ535_PN_In_Out_32_byte_1[21] := HwInputs.ST80_1_TZ535_PN_In_Out_32_byte_1[21];
	PlcInputs.ST80_1_TZ535_PN_In_Out_32_byte_1[22] := HwInputs.ST80_1_TZ535_PN_In_Out_32_byte_1[22];
	PlcInputs.ST80_1_TZ535_PN_In_Out_32_byte_1[23] := HwInputs.ST80_1_TZ535_PN_In_Out_32_byte_1[23];
	PlcInputs.ST80_1_TZ535_PN_In_Out_32_byte_1[24] := HwInputs.ST80_1_TZ535_PN_In_Out_32_byte_1[24];
	PlcInputs.ST80_1_TZ535_PN_In_Out_32_byte_1[25] := HwInputs.ST80_1_TZ535_PN_In_Out_32_byte_1[25];
	PlcInputs.ST80_1_TZ535_PN_In_Out_32_byte_1[26] := HwInputs.ST80_1_TZ535_PN_In_Out_32_byte_1[26];
	PlcInputs.ST80_1_TZ535_PN_In_Out_32_byte_1[27] := HwInputs.ST80_1_TZ535_PN_In_Out_32_byte_1[27];
	PlcInputs.ST80_1_TZ535_PN_In_Out_32_byte_1[28] := HwInputs.ST80_1_TZ535_PN_In_Out_32_byte_1[28];
	PlcInputs.ST80_1_TZ535_PN_In_Out_32_byte_1[29] := HwInputs.ST80_1_TZ535_PN_In_Out_32_byte_1[29];
	PlcInputs.ST80_1_TZ535_PN_In_Out_32_byte_1[30] := HwInputs.ST80_1_TZ535_PN_In_Out_32_byte_1[30];
	PlcInputs.ST80_1_TZ535_PN_In_Out_32_byte_1[31] := HwInputs.ST80_1_TZ535_PN_In_Out_32_byte_1[31];
	PlcInputs.ST80_1_DM260_Housing_Acquisition_Status_1[0] := HwInputs.ST80_1_DM260_Housing_Acquisition_Status_1[0];
	PlcInputs.ST80_1_DM260_Housing_Acquisition_Status_1[1] := HwInputs.ST80_1_DM260_Housing_Acquisition_Status_1[1];
	PlcInputs.ST80_1_DM260_Housing_Acquisition_Status_1[2] := HwInputs.ST80_1_DM260_Housing_Acquisition_Status_1[2];
	PlcInputs.ST80_1_DM260_Housing_Results_Status_1 := HwInputs.ST80_1_DM260_Housing_Results_Status_1;
	PlcInputs.ST80_1_DM260_Housing_Soft_Event_Control_1 := HwInputs.ST80_1_DM260_Housing_Soft_Event_Control_1;
	PlcInputs.ST80_1_DM260_Housing_Result_Data_64_bytes_1[0] := HwInputs.ST80_1_DM260_Housing_Result_Data_64_bytes_1[0];
	PlcInputs.ST80_1_DM260_Housing_Result_Data_64_bytes_1[1] := HwInputs.ST80_1_DM260_Housing_Result_Data_64_bytes_1[1];
	PlcInputs.ST80_1_DM260_Housing_Result_Data_64_bytes_1[2] := HwInputs.ST80_1_DM260_Housing_Result_Data_64_bytes_1[2];
	PlcInputs.ST80_1_DM260_Housing_Result_Data_64_bytes_1[3] := HwInputs.ST80_1_DM260_Housing_Result_Data_64_bytes_1[3];
	PlcInputs.ST80_1_DM260_Housing_Result_Data_64_bytes_1[4] := HwInputs.ST80_1_DM260_Housing_Result_Data_64_bytes_1[4];
	PlcInputs.ST80_1_DM260_Housing_Result_Data_64_bytes_1[5] := HwInputs.ST80_1_DM260_Housing_Result_Data_64_bytes_1[5];
	PlcInputs.ST80_1_DM260_Housing_Result_Data_64_bytes_1[6] := HwInputs.ST80_1_DM260_Housing_Result_Data_64_bytes_1[6];
	PlcInputs.ST80_1_DM260_Housing_Result_Data_64_bytes_1[7] := HwInputs.ST80_1_DM260_Housing_Result_Data_64_bytes_1[7];
	PlcInputs.ST80_1_DM260_Housing_Result_Data_64_bytes_1[8] := HwInputs.ST80_1_DM260_Housing_Result_Data_64_bytes_1[8];
	PlcInputs.ST80_1_DM260_Housing_Result_Data_64_bytes_1[9] := HwInputs.ST80_1_DM260_Housing_Result_Data_64_bytes_1[9];
	PlcInputs.ST80_1_DM260_Housing_Result_Data_64_bytes_1[10] := HwInputs.ST80_1_DM260_Housing_Result_Data_64_bytes_1[10];
	PlcInputs.ST80_1_DM260_Housing_Result_Data_64_bytes_1[11] := HwInputs.ST80_1_DM260_Housing_Result_Data_64_bytes_1[11];
	PlcInputs.ST80_1_DM260_Housing_Result_Data_64_bytes_1[12] := HwInputs.ST80_1_DM260_Housing_Result_Data_64_bytes_1[12];
	PlcInputs.ST80_1_DM260_Housing_Result_Data_64_bytes_1[13] := HwInputs.ST80_1_DM260_Housing_Result_Data_64_bytes_1[13];
	PlcInputs.ST80_1_DM260_Housing_Result_Data_64_bytes_1[14] := HwInputs.ST80_1_DM260_Housing_Result_Data_64_bytes_1[14];
	PlcInputs.ST80_1_DM260_Housing_Result_Data_64_bytes_1[15] := HwInputs.ST80_1_DM260_Housing_Result_Data_64_bytes_1[15];
	PlcInputs.ST80_1_DM260_Housing_Result_Data_64_bytes_1[16] := HwInputs.ST80_1_DM260_Housing_Result_Data_64_bytes_1[16];
	PlcInputs.ST80_1_DM260_Housing_Result_Data_64_bytes_1[17] := HwInputs.ST80_1_DM260_Housing_Result_Data_64_bytes_1[17];
	PlcInputs.ST80_1_DM260_Housing_Result_Data_64_bytes_1[18] := HwInputs.ST80_1_DM260_Housing_Result_Data_64_bytes_1[18];
	PlcInputs.ST80_1_DM260_Housing_Result_Data_64_bytes_1[19] := HwInputs.ST80_1_DM260_Housing_Result_Data_64_bytes_1[19];
	PlcInputs.ST80_1_DM260_Housing_Result_Data_64_bytes_1[20] := HwInputs.ST80_1_DM260_Housing_Result_Data_64_bytes_1[20];
	PlcInputs.ST80_1_DM260_Housing_Result_Data_64_bytes_1[21] := HwInputs.ST80_1_DM260_Housing_Result_Data_64_bytes_1[21];
	PlcInputs.ST80_1_DM260_Housing_Result_Data_64_bytes_1[22] := HwInputs.ST80_1_DM260_Housing_Result_Data_64_bytes_1[22];
	PlcInputs.ST80_1_DM260_Housing_Result_Data_64_bytes_1[23] := HwInputs.ST80_1_DM260_Housing_Result_Data_64_bytes_1[23];
	PlcInputs.ST80_1_DM260_Housing_Result_Data_64_bytes_1[24] := HwInputs.ST80_1_DM260_Housing_Result_Data_64_bytes_1[24];
	PlcInputs.ST80_1_DM260_Housing_Result_Data_64_bytes_1[25] := HwInputs.ST80_1_DM260_Housing_Result_Data_64_bytes_1[25];
	PlcInputs.ST80_1_DM260_Housing_Result_Data_64_bytes_1[26] := HwInputs.ST80_1_DM260_Housing_Result_Data_64_bytes_1[26];
	PlcInputs.ST80_1_DM260_Housing_Result_Data_64_bytes_1[27] := HwInputs.ST80_1_DM260_Housing_Result_Data_64_bytes_1[27];
	PlcInputs.ST80_1_DM260_Housing_Result_Data_64_bytes_1[28] := HwInputs.ST80_1_DM260_Housing_Result_Data_64_bytes_1[28];
	PlcInputs.ST80_1_DM260_Housing_Result_Data_64_bytes_1[29] := HwInputs.ST80_1_DM260_Housing_Result_Data_64_bytes_1[29];
	PlcInputs.ST80_1_DM260_Housing_Result_Data_64_bytes_1[30] := HwInputs.ST80_1_DM260_Housing_Result_Data_64_bytes_1[30];
	PlcInputs.ST80_1_DM260_Housing_Result_Data_64_bytes_1[31] := HwInputs.ST80_1_DM260_Housing_Result_Data_64_bytes_1[31];
	PlcInputs.ST80_1_DM260_Housing_Result_Data_64_bytes_1[32] := HwInputs.ST80_1_DM260_Housing_Result_Data_64_bytes_1[32];
	PlcInputs.ST80_1_DM260_Housing_Result_Data_64_bytes_1[33] := HwInputs.ST80_1_DM260_Housing_Result_Data_64_bytes_1[33];
	PlcInputs.ST80_1_DM260_Housing_Result_Data_64_bytes_1[34] := HwInputs.ST80_1_DM260_Housing_Result_Data_64_bytes_1[34];
	PlcInputs.ST80_1_DM260_Housing_Result_Data_64_bytes_1[35] := HwInputs.ST80_1_DM260_Housing_Result_Data_64_bytes_1[35];
	PlcInputs.ST80_1_DM260_Housing_Result_Data_64_bytes_1[36] := HwInputs.ST80_1_DM260_Housing_Result_Data_64_bytes_1[36];
	PlcInputs.ST80_1_DM260_Housing_Result_Data_64_bytes_1[37] := HwInputs.ST80_1_DM260_Housing_Result_Data_64_bytes_1[37];
	PlcInputs.ST80_1_DM260_Housing_Result_Data_64_bytes_1[38] := HwInputs.ST80_1_DM260_Housing_Result_Data_64_bytes_1[38];
	PlcInputs.ST80_1_DM260_Housing_Result_Data_64_bytes_1[39] := HwInputs.ST80_1_DM260_Housing_Result_Data_64_bytes_1[39];
	PlcInputs.ST80_1_DM260_Housing_Result_Data_64_bytes_1[40] := HwInputs.ST80_1_DM260_Housing_Result_Data_64_bytes_1[40];
	PlcInputs.ST80_1_DM260_Housing_Result_Data_64_bytes_1[41] := HwInputs.ST80_1_DM260_Housing_Result_Data_64_bytes_1[41];
	PlcInputs.ST80_1_DM260_Housing_Result_Data_64_bytes_1[42] := HwInputs.ST80_1_DM260_Housing_Result_Data_64_bytes_1[42];
	PlcInputs.ST80_1_DM260_Housing_Result_Data_64_bytes_1[43] := HwInputs.ST80_1_DM260_Housing_Result_Data_64_bytes_1[43];
	PlcInputs.ST80_1_DM260_Housing_Result_Data_64_bytes_1[44] := HwInputs.ST80_1_DM260_Housing_Result_Data_64_bytes_1[44];
	PlcInputs.ST80_1_DM260_Housing_Result_Data_64_bytes_1[45] := HwInputs.ST80_1_DM260_Housing_Result_Data_64_bytes_1[45];
	PlcInputs.ST80_1_DM260_Housing_Result_Data_64_bytes_1[46] := HwInputs.ST80_1_DM260_Housing_Result_Data_64_bytes_1[46];
	PlcInputs.ST80_1_DM260_Housing_Result_Data_64_bytes_1[47] := HwInputs.ST80_1_DM260_Housing_Result_Data_64_bytes_1[47];
	PlcInputs.ST80_1_DM260_Housing_Result_Data_64_bytes_1[48] := HwInputs.ST80_1_DM260_Housing_Result_Data_64_bytes_1[48];
	PlcInputs.ST80_1_DM260_Housing_Result_Data_64_bytes_1[49] := HwInputs.ST80_1_DM260_Housing_Result_Data_64_bytes_1[49];
	PlcInputs.ST80_1_DM260_Housing_Result_Data_64_bytes_1[50] := HwInputs.ST80_1_DM260_Housing_Result_Data_64_bytes_1[50];
	PlcInputs.ST80_1_DM260_Housing_Result_Data_64_bytes_1[51] := HwInputs.ST80_1_DM260_Housing_Result_Data_64_bytes_1[51];
	PlcInputs.ST80_1_DM260_Housing_Result_Data_64_bytes_1[52] := HwInputs.ST80_1_DM260_Housing_Result_Data_64_bytes_1[52];
	PlcInputs.ST80_1_DM260_Housing_Result_Data_64_bytes_1[53] := HwInputs.ST80_1_DM260_Housing_Result_Data_64_bytes_1[53];
	PlcInputs.ST80_1_DM260_Housing_Result_Data_64_bytes_1[54] := HwInputs.ST80_1_DM260_Housing_Result_Data_64_bytes_1[54];
	PlcInputs.ST80_1_DM260_Housing_Result_Data_64_bytes_1[55] := HwInputs.ST80_1_DM260_Housing_Result_Data_64_bytes_1[55];
	PlcInputs.ST80_1_DM260_Housing_Result_Data_64_bytes_1[56] := HwInputs.ST80_1_DM260_Housing_Result_Data_64_bytes_1[56];
	PlcInputs.ST80_1_DM260_Housing_Result_Data_64_bytes_1[57] := HwInputs.ST80_1_DM260_Housing_Result_Data_64_bytes_1[57];
	PlcInputs.ST80_1_DM260_Housing_Result_Data_64_bytes_1[58] := HwInputs.ST80_1_DM260_Housing_Result_Data_64_bytes_1[58];
	PlcInputs.ST80_1_DM260_Housing_Result_Data_64_bytes_1[59] := HwInputs.ST80_1_DM260_Housing_Result_Data_64_bytes_1[59];
	PlcInputs.ST80_1_DM260_Housing_Result_Data_64_bytes_1[60] := HwInputs.ST80_1_DM260_Housing_Result_Data_64_bytes_1[60];
	PlcInputs.ST80_1_DM260_Housing_Result_Data_64_bytes_1[61] := HwInputs.ST80_1_DM260_Housing_Result_Data_64_bytes_1[61];
	PlcInputs.ST80_1_DM260_Housing_Result_Data_64_bytes_1[62] := HwInputs.ST80_1_DM260_Housing_Result_Data_64_bytes_1[62];
	PlcInputs.ST80_1_DM260_Housing_Result_Data_64_bytes_1[63] := HwInputs.ST80_1_DM260_Housing_Result_Data_64_bytes_1[63];
	PlcInputs.ST80_1_DM260_Housing_Result_Data_64_bytes_1[64] := HwInputs.ST80_1_DM260_Housing_Result_Data_64_bytes_1[64];
	PlcInputs.ST80_1_DM260_Housing_Result_Data_64_bytes_1[65] := HwInputs.ST80_1_DM260_Housing_Result_Data_64_bytes_1[65];
	PlcInputs.ST80_1_DM260_Housing_Result_Data_64_bytes_1[66] := HwInputs.ST80_1_DM260_Housing_Result_Data_64_bytes_1[66];
	PlcInputs.ST80_1_DM260_Housing_Result_Data_64_bytes_1[67] := HwInputs.ST80_1_DM260_Housing_Result_Data_64_bytes_1[67];
	PlcInputs.ST80_1_DM260_Housing_Result_Data_64_bytes_1[68] := HwInputs.ST80_1_DM260_Housing_Result_Data_64_bytes_1[68];
	PlcInputs.ST80_1_DM260_Housing_Result_Data_64_bytes_1[69] := HwInputs.ST80_1_DM260_Housing_Result_Data_64_bytes_1[69];
	PlcInputs.ST80_1_DM260_Housing_Result_Data_64_bytes_1[70] := HwInputs.ST80_1_DM260_Housing_Result_Data_64_bytes_1[70];
	PlcInputs.ST80_1_DM260_Housing_Result_Data_64_bytes_1[71] := HwInputs.ST80_1_DM260_Housing_Result_Data_64_bytes_1[71];
	PlcInputs.ST80_ET200SP_CM_4xIO_Link_1[0] := HwInputs.ST80_ET200SP_CM_4xIO_Link_1[0];
	PlcInputs.ST80_ET200SP_CM_4xIO_Link_1[1] := HwInputs.ST80_ET200SP_CM_4xIO_Link_1[1];
	PlcInputs.ST80_ET200SP_CM_4xIO_Link_1[2] := HwInputs.ST80_ET200SP_CM_4xIO_Link_1[2];
	PlcInputs.ST80_ET200SP_CM_4xIO_Link_1[3] := HwInputs.ST80_ET200SP_CM_4xIO_Link_1[3];
	PlcInputs.ST80_ET200SP_CM_4xIO_Link_1[4] := HwInputs.ST80_ET200SP_CM_4xIO_Link_1[4];
	PlcInputs.ST80_ET200SP_CM_4xIO_Link_1[5] := HwInputs.ST80_ET200SP_CM_4xIO_Link_1[5];
	PlcInputs.ST80_ET200SP_CM_4xIO_Link_1[6] := HwInputs.ST80_ET200SP_CM_4xIO_Link_1[6];
	PlcInputs.ST80_ET200SP_CM_4xIO_Link_1[7] := HwInputs.ST80_ET200SP_CM_4xIO_Link_1[7];
	PlcInputs.ST80_ET200SP_CM_4xIO_Link_1[8] := HwInputs.ST80_ET200SP_CM_4xIO_Link_1[8];
	PlcInputs.ST80_ET200SP_CM_4xIO_Link_1[9] := HwInputs.ST80_ET200SP_CM_4xIO_Link_1[9];
	PlcInputs.ST80_ET200SP_CM_4xIO_Link_1[10] := HwInputs.ST80_ET200SP_CM_4xIO_Link_1[10];
	PlcInputs.ST80_ET200SP_CM_4xIO_Link_1[11] := HwInputs.ST80_ET200SP_CM_4xIO_Link_1[11];
	PlcInputs.ST80_ET200SP_CM_4xIO_Link_1[12] := HwInputs.ST80_ET200SP_CM_4xIO_Link_1[12];
	PlcInputs.ST80_ET200SP_CM_4xIO_Link_1[13] := HwInputs.ST80_ET200SP_CM_4xIO_Link_1[13];
	PlcInputs.ST80_ET200SP_CM_4xIO_Link_1[14] := HwInputs.ST80_ET200SP_CM_4xIO_Link_1[14];
	PlcInputs.ST80_ET200SP_CM_4xIO_Link_1[15] := HwInputs.ST80_ET200SP_CM_4xIO_Link_1[15];
	PlcInputs.ST80_ET200SP_CM_4xIO_Link_1[16] := HwInputs.ST80_ET200SP_CM_4xIO_Link_1[16];
	PlcInputs.ST80_ET200SP_CM_4xIO_Link_1[17] := HwInputs.ST80_ET200SP_CM_4xIO_Link_1[17];
	PlcInputs.ST80_ET200SP_CM_4xIO_Link_1[18] := HwInputs.ST80_ET200SP_CM_4xIO_Link_1[18];
	PlcInputs.ST80_ET200SP_CM_4xIO_Link_1[19] := HwInputs.ST80_ET200SP_CM_4xIO_Link_1[19];
	PlcInputs.ST80_ET200SP_CM_4xIO_Link_1[20] := HwInputs.ST80_ET200SP_CM_4xIO_Link_1[20];
	PlcInputs.ST80_ET200SP_CM_4xIO_Link_1[21] := HwInputs.ST80_ET200SP_CM_4xIO_Link_1[21];
	PlcInputs.ST80_ET200SP_CM_4xIO_Link_1[22] := HwInputs.ST80_ET200SP_CM_4xIO_Link_1[22];
	PlcInputs.ST80_ET200SP_CM_4xIO_Link_1[23] := HwInputs.ST80_ET200SP_CM_4xIO_Link_1[23];
	PlcInputs.ST80_ET200SP_CM_4xIO_Link_1[24] := HwInputs.ST80_ET200SP_CM_4xIO_Link_1[24];
	PlcInputs.ST80_ET200SP_CM_4xIO_Link_1[25] := HwInputs.ST80_ET200SP_CM_4xIO_Link_1[25];
	PlcInputs.ST80_ET200SP_CM_4xIO_Link_1[26] := HwInputs.ST80_ET200SP_CM_4xIO_Link_1[26];
	PlcInputs.ST80_ET200SP_CM_4xIO_Link_1[27] := HwInputs.ST80_ET200SP_CM_4xIO_Link_1[27];
	PlcInputs.ST80_ET200SP_CM_4xIO_Link_1[28] := HwInputs.ST80_ET200SP_CM_4xIO_Link_1[28];
	PlcInputs.ST80_ET200SP_CM_4xIO_Link_1[29] := HwInputs.ST80_ET200SP_CM_4xIO_Link_1[29];
	PlcInputs.ST80_ET200SP_CM_4xIO_Link_1[30] := HwInputs.ST80_ET200SP_CM_4xIO_Link_1[30];
	PlcInputs.ST80_ET200SP_CM_4xIO_Link_1[31] := HwInputs.ST80_ET200SP_CM_4xIO_Link_1[31];
	PlcInputs.ST80_ET200SP_CM_4xIO_Link_2[0] := HwInputs.ST80_ET200SP_CM_4xIO_Link_2[0];
	PlcInputs.ST80_ET200SP_CM_4xIO_Link_2[1] := HwInputs.ST80_ET200SP_CM_4xIO_Link_2[1];
	PlcInputs.ST80_ET200SP_CM_4xIO_Link_2[2] := HwInputs.ST80_ET200SP_CM_4xIO_Link_2[2];
	PlcInputs.ST80_ET200SP_CM_4xIO_Link_2[3] := HwInputs.ST80_ET200SP_CM_4xIO_Link_2[3];
	PlcInputs.ST80_ET200SP_CM_4xIO_Link_2[4] := HwInputs.ST80_ET200SP_CM_4xIO_Link_2[4];
	PlcInputs.ST80_ET200SP_CM_4xIO_Link_2[5] := HwInputs.ST80_ET200SP_CM_4xIO_Link_2[5];
	PlcInputs.ST80_ET200SP_CM_4xIO_Link_2[6] := HwInputs.ST80_ET200SP_CM_4xIO_Link_2[6];
	PlcInputs.ST80_ET200SP_CM_4xIO_Link_2[7] := HwInputs.ST80_ET200SP_CM_4xIO_Link_2[7];
	PlcInputs.ST80_ET200SP_CM_4xIO_Link_2[8] := HwInputs.ST80_ET200SP_CM_4xIO_Link_2[8];
	PlcInputs.ST80_ET200SP_CM_4xIO_Link_2[9] := HwInputs.ST80_ET200SP_CM_4xIO_Link_2[9];
	PlcInputs.ST80_ET200SP_CM_4xIO_Link_2[10] := HwInputs.ST80_ET200SP_CM_4xIO_Link_2[10];
	PlcInputs.ST80_ET200SP_CM_4xIO_Link_2[11] := HwInputs.ST80_ET200SP_CM_4xIO_Link_2[11];
	PlcInputs.ST80_ET200SP_CM_4xIO_Link_2[12] := HwInputs.ST80_ET200SP_CM_4xIO_Link_2[12];
	PlcInputs.ST80_ET200SP_CM_4xIO_Link_2[13] := HwInputs.ST80_ET200SP_CM_4xIO_Link_2[13];
	PlcInputs.ST80_ET200SP_CM_4xIO_Link_2[14] := HwInputs.ST80_ET200SP_CM_4xIO_Link_2[14];
	PlcInputs.ST80_ET200SP_CM_4xIO_Link_2[15] := HwInputs.ST80_ET200SP_CM_4xIO_Link_2[15];
	PlcInputs.ST80_ET200SP_CM_4xIO_Link_2[16] := HwInputs.ST80_ET200SP_CM_4xIO_Link_2[16];
	PlcInputs.ST80_ET200SP_CM_4xIO_Link_2[17] := HwInputs.ST80_ET200SP_CM_4xIO_Link_2[17];
	PlcInputs.ST80_ET200SP_CM_4xIO_Link_2[18] := HwInputs.ST80_ET200SP_CM_4xIO_Link_2[18];
	PlcInputs.ST80_ET200SP_CM_4xIO_Link_2[19] := HwInputs.ST80_ET200SP_CM_4xIO_Link_2[19];
	PlcInputs.ST80_ET200SP_CM_4xIO_Link_2[20] := HwInputs.ST80_ET200SP_CM_4xIO_Link_2[20];
	PlcInputs.ST80_ET200SP_CM_4xIO_Link_2[21] := HwInputs.ST80_ET200SP_CM_4xIO_Link_2[21];
	PlcInputs.ST80_ET200SP_CM_4xIO_Link_2[22] := HwInputs.ST80_ET200SP_CM_4xIO_Link_2[22];
	PlcInputs.ST80_ET200SP_CM_4xIO_Link_2[23] := HwInputs.ST80_ET200SP_CM_4xIO_Link_2[23];
	PlcInputs.ST80_ET200SP_CM_4xIO_Link_2[24] := HwInputs.ST80_ET200SP_CM_4xIO_Link_2[24];
	PlcInputs.ST80_ET200SP_CM_4xIO_Link_2[25] := HwInputs.ST80_ET200SP_CM_4xIO_Link_2[25];
	PlcInputs.ST80_ET200SP_CM_4xIO_Link_2[26] := HwInputs.ST80_ET200SP_CM_4xIO_Link_2[26];
	PlcInputs.ST80_ET200SP_CM_4xIO_Link_2[27] := HwInputs.ST80_ET200SP_CM_4xIO_Link_2[27];
	PlcInputs.ST80_ET200SP_CM_4xIO_Link_2[28] := HwInputs.ST80_ET200SP_CM_4xIO_Link_2[28];
	PlcInputs.ST80_ET200SP_CM_4xIO_Link_2[29] := HwInputs.ST80_ET200SP_CM_4xIO_Link_2[29];
	PlcInputs.ST80_ET200SP_CM_4xIO_Link_2[30] := HwInputs.ST80_ET200SP_CM_4xIO_Link_2[30];
	PlcInputs.ST80_ET200SP_CM_4xIO_Link_2[31] := HwInputs.ST80_ET200SP_CM_4xIO_Link_2[31];
	PlcInputs.ST80_ET200SP_CM_4xIO_Link_3[0] := HwInputs.ST80_ET200SP_CM_4xIO_Link_3[0];
	PlcInputs.ST80_ET200SP_CM_4xIO_Link_3[1] := HwInputs.ST80_ET200SP_CM_4xIO_Link_3[1];
	PlcInputs.ST80_ET200SP_CM_4xIO_Link_3[2] := HwInputs.ST80_ET200SP_CM_4xIO_Link_3[2];
	PlcInputs.ST80_ET200SP_CM_4xIO_Link_3[3] := HwInputs.ST80_ET200SP_CM_4xIO_Link_3[3];
	PlcInputs.ST80_ET200SP_CM_4xIO_Link_3[4] := HwInputs.ST80_ET200SP_CM_4xIO_Link_3[4];
	PlcInputs.ST80_ET200SP_CM_4xIO_Link_3[5] := HwInputs.ST80_ET200SP_CM_4xIO_Link_3[5];
	PlcInputs.ST80_ET200SP_CM_4xIO_Link_3[6] := HwInputs.ST80_ET200SP_CM_4xIO_Link_3[6];
	PlcInputs.ST80_ET200SP_CM_4xIO_Link_3[7] := HwInputs.ST80_ET200SP_CM_4xIO_Link_3[7];
	PlcInputs.ST80_ET200SP_CM_4xIO_Link_3[8] := HwInputs.ST80_ET200SP_CM_4xIO_Link_3[8];
	PlcInputs.ST80_ET200SP_CM_4xIO_Link_3[9] := HwInputs.ST80_ET200SP_CM_4xIO_Link_3[9];
	PlcInputs.ST80_ET200SP_CM_4xIO_Link_3[10] := HwInputs.ST80_ET200SP_CM_4xIO_Link_3[10];
	PlcInputs.ST80_ET200SP_CM_4xIO_Link_3[11] := HwInputs.ST80_ET200SP_CM_4xIO_Link_3[11];
	PlcInputs.ST80_ET200SP_CM_4xIO_Link_3[12] := HwInputs.ST80_ET200SP_CM_4xIO_Link_3[12];
	PlcInputs.ST80_ET200SP_CM_4xIO_Link_3[13] := HwInputs.ST80_ET200SP_CM_4xIO_Link_3[13];
	PlcInputs.ST80_ET200SP_CM_4xIO_Link_3[14] := HwInputs.ST80_ET200SP_CM_4xIO_Link_3[14];
	PlcInputs.ST80_ET200SP_CM_4xIO_Link_3[15] := HwInputs.ST80_ET200SP_CM_4xIO_Link_3[15];
	PlcInputs.ST80_ET200SP_CM_4xIO_Link_3[16] := HwInputs.ST80_ET200SP_CM_4xIO_Link_3[16];
	PlcInputs.ST80_ET200SP_CM_4xIO_Link_3[17] := HwInputs.ST80_ET200SP_CM_4xIO_Link_3[17];
	PlcInputs.ST80_ET200SP_CM_4xIO_Link_3[18] := HwInputs.ST80_ET200SP_CM_4xIO_Link_3[18];
	PlcInputs.ST80_ET200SP_CM_4xIO_Link_3[19] := HwInputs.ST80_ET200SP_CM_4xIO_Link_3[19];
	PlcInputs.ST80_ET200SP_CM_4xIO_Link_3[20] := HwInputs.ST80_ET200SP_CM_4xIO_Link_3[20];
	PlcInputs.ST80_ET200SP_CM_4xIO_Link_3[21] := HwInputs.ST80_ET200SP_CM_4xIO_Link_3[21];
	PlcInputs.ST80_ET200SP_CM_4xIO_Link_3[22] := HwInputs.ST80_ET200SP_CM_4xIO_Link_3[22];
	PlcInputs.ST80_ET200SP_CM_4xIO_Link_3[23] := HwInputs.ST80_ET200SP_CM_4xIO_Link_3[23];
	PlcInputs.ST80_ET200SP_CM_4xIO_Link_3[24] := HwInputs.ST80_ET200SP_CM_4xIO_Link_3[24];
	PlcInputs.ST80_ET200SP_CM_4xIO_Link_3[25] := HwInputs.ST80_ET200SP_CM_4xIO_Link_3[25];
	PlcInputs.ST80_ET200SP_CM_4xIO_Link_3[26] := HwInputs.ST80_ET200SP_CM_4xIO_Link_3[26];
	PlcInputs.ST80_ET200SP_CM_4xIO_Link_3[27] := HwInputs.ST80_ET200SP_CM_4xIO_Link_3[27];
	PlcInputs.ST80_ET200SP_CM_4xIO_Link_3[28] := HwInputs.ST80_ET200SP_CM_4xIO_Link_3[28];
	PlcInputs.ST80_ET200SP_CM_4xIO_Link_3[29] := HwInputs.ST80_ET200SP_CM_4xIO_Link_3[29];
	PlcInputs.ST80_ET200SP_CM_4xIO_Link_3[30] := HwInputs.ST80_ET200SP_CM_4xIO_Link_3[30];
	PlcInputs.ST80_ET200SP_CM_4xIO_Link_3[31] := HwInputs.ST80_ET200SP_CM_4xIO_Link_3[31];
	PlcInputs.ST80_ET200SP_DI_16x24VDC_ST_1 := HwInputs.ST80_ET200SP_DI_16x24VDC_ST_1;
	PlcInputs.ST80_ET200SP_DI_16x24VDC_ST_2 := HwInputs.ST80_ET200SP_DI_16x24VDC_ST_2;
	PlcInputs.ST80_ET200SP_DI_16x24VDC_ST_3 := HwInputs.ST80_ET200SP_DI_16x24VDC_ST_3;
	PlcInputs.ST80_ET200SP_DI_16x24VDC_ST_4 := HwInputs.ST80_ET200SP_DI_16x24VDC_ST_4;
END_FUNCTION

(* ---- CopyOutputs.st ---- *)
FUNCTION CopyOutputs
	VAR_EXTERNAL
		HwOutputs : HwOutputs;
		PlcOutputs : PlcOutputs;
	END_VAR
	HwOutputs.ST80_1_DM260_EB_Box_Acquisition_Control_1 := PlcOutputs.ST80_1_DM260_EB_Box_Acquisition_Control_1;
	HwOutputs.ST80_1_DM260_EB_Box_Results_Control_1 := PlcOutputs.ST80_1_DM260_EB_Box_Results_Control_1;
	HwOutputs.ST80_1_DM260_EB_Box_Soft_Event_Control_1 := PlcOutputs.ST80_1_DM260_EB_Box_Soft_Event_Control_1;
	HwOutputs.ST80_1_DM260_EB_Box_User_Data_64_bytes_1[0] := PlcOutputs.ST80_1_DM260_EB_Box_User_Data_64_bytes_1[0];
	HwOutputs.ST80_1_DM260_EB_Box_User_Data_64_bytes_1[1] := PlcOutputs.ST80_1_DM260_EB_Box_User_Data_64_bytes_1[1];
	HwOutputs.ST80_1_DM260_EB_Box_User_Data_64_bytes_1[2] := PlcOutputs.ST80_1_DM260_EB_Box_User_Data_64_bytes_1[2];
	HwOutputs.ST80_1_DM260_EB_Box_User_Data_64_bytes_1[3] := PlcOutputs.ST80_1_DM260_EB_Box_User_Data_64_bytes_1[3];
	HwOutputs.ST80_1_DM260_EB_Box_User_Data_64_bytes_1[4] := PlcOutputs.ST80_1_DM260_EB_Box_User_Data_64_bytes_1[4];
	HwOutputs.ST80_1_DM260_EB_Box_User_Data_64_bytes_1[5] := PlcOutputs.ST80_1_DM260_EB_Box_User_Data_64_bytes_1[5];
	HwOutputs.ST80_1_DM260_EB_Box_User_Data_64_bytes_1[6] := PlcOutputs.ST80_1_DM260_EB_Box_User_Data_64_bytes_1[6];
	HwOutputs.ST80_1_DM260_EB_Box_User_Data_64_bytes_1[7] := PlcOutputs.ST80_1_DM260_EB_Box_User_Data_64_bytes_1[7];
	HwOutputs.ST80_1_DM260_EB_Box_User_Data_64_bytes_1[8] := PlcOutputs.ST80_1_DM260_EB_Box_User_Data_64_bytes_1[8];
	HwOutputs.ST80_1_DM260_EB_Box_User_Data_64_bytes_1[9] := PlcOutputs.ST80_1_DM260_EB_Box_User_Data_64_bytes_1[9];
	HwOutputs.ST80_1_DM260_EB_Box_User_Data_64_bytes_1[10] := PlcOutputs.ST80_1_DM260_EB_Box_User_Data_64_bytes_1[10];
	HwOutputs.ST80_1_DM260_EB_Box_User_Data_64_bytes_1[11] := PlcOutputs.ST80_1_DM260_EB_Box_User_Data_64_bytes_1[11];
	HwOutputs.ST80_1_DM260_EB_Box_User_Data_64_bytes_1[12] := PlcOutputs.ST80_1_DM260_EB_Box_User_Data_64_bytes_1[12];
	HwOutputs.ST80_1_DM260_EB_Box_User_Data_64_bytes_1[13] := PlcOutputs.ST80_1_DM260_EB_Box_User_Data_64_bytes_1[13];
	HwOutputs.ST80_1_DM260_EB_Box_User_Data_64_bytes_1[14] := PlcOutputs.ST80_1_DM260_EB_Box_User_Data_64_bytes_1[14];
	HwOutputs.ST80_1_DM260_EB_Box_User_Data_64_bytes_1[15] := PlcOutputs.ST80_1_DM260_EB_Box_User_Data_64_bytes_1[15];
	HwOutputs.ST80_1_DM260_EB_Box_User_Data_64_bytes_1[16] := PlcOutputs.ST80_1_DM260_EB_Box_User_Data_64_bytes_1[16];
	HwOutputs.ST80_1_DM260_EB_Box_User_Data_64_bytes_1[17] := PlcOutputs.ST80_1_DM260_EB_Box_User_Data_64_bytes_1[17];
	HwOutputs.ST80_1_DM260_EB_Box_User_Data_64_bytes_1[18] := PlcOutputs.ST80_1_DM260_EB_Box_User_Data_64_bytes_1[18];
	HwOutputs.ST80_1_DM260_EB_Box_User_Data_64_bytes_1[19] := PlcOutputs.ST80_1_DM260_EB_Box_User_Data_64_bytes_1[19];
	HwOutputs.ST80_1_DM260_EB_Box_User_Data_64_bytes_1[20] := PlcOutputs.ST80_1_DM260_EB_Box_User_Data_64_bytes_1[20];
	HwOutputs.ST80_1_DM260_EB_Box_User_Data_64_bytes_1[21] := PlcOutputs.ST80_1_DM260_EB_Box_User_Data_64_bytes_1[21];
	HwOutputs.ST80_1_DM260_EB_Box_User_Data_64_bytes_1[22] := PlcOutputs.ST80_1_DM260_EB_Box_User_Data_64_bytes_1[22];
	HwOutputs.ST80_1_DM260_EB_Box_User_Data_64_bytes_1[23] := PlcOutputs.ST80_1_DM260_EB_Box_User_Data_64_bytes_1[23];
	HwOutputs.ST80_1_DM260_EB_Box_User_Data_64_bytes_1[24] := PlcOutputs.ST80_1_DM260_EB_Box_User_Data_64_bytes_1[24];
	HwOutputs.ST80_1_DM260_EB_Box_User_Data_64_bytes_1[25] := PlcOutputs.ST80_1_DM260_EB_Box_User_Data_64_bytes_1[25];
	HwOutputs.ST80_1_DM260_EB_Box_User_Data_64_bytes_1[26] := PlcOutputs.ST80_1_DM260_EB_Box_User_Data_64_bytes_1[26];
	HwOutputs.ST80_1_DM260_EB_Box_User_Data_64_bytes_1[27] := PlcOutputs.ST80_1_DM260_EB_Box_User_Data_64_bytes_1[27];
	HwOutputs.ST80_1_DM260_EB_Box_User_Data_64_bytes_1[28] := PlcOutputs.ST80_1_DM260_EB_Box_User_Data_64_bytes_1[28];
	HwOutputs.ST80_1_DM260_EB_Box_User_Data_64_bytes_1[29] := PlcOutputs.ST80_1_DM260_EB_Box_User_Data_64_bytes_1[29];
	HwOutputs.ST80_1_DM260_EB_Box_User_Data_64_bytes_1[30] := PlcOutputs.ST80_1_DM260_EB_Box_User_Data_64_bytes_1[30];
	HwOutputs.ST80_1_DM260_EB_Box_User_Data_64_bytes_1[31] := PlcOutputs.ST80_1_DM260_EB_Box_User_Data_64_bytes_1[31];
	HwOutputs.ST80_1_DM260_EB_Box_User_Data_64_bytes_1[32] := PlcOutputs.ST80_1_DM260_EB_Box_User_Data_64_bytes_1[32];
	HwOutputs.ST80_1_DM260_EB_Box_User_Data_64_bytes_1[33] := PlcOutputs.ST80_1_DM260_EB_Box_User_Data_64_bytes_1[33];
	HwOutputs.ST80_1_DM260_EB_Box_User_Data_64_bytes_1[34] := PlcOutputs.ST80_1_DM260_EB_Box_User_Data_64_bytes_1[34];
	HwOutputs.ST80_1_DM260_EB_Box_User_Data_64_bytes_1[35] := PlcOutputs.ST80_1_DM260_EB_Box_User_Data_64_bytes_1[35];
	HwOutputs.ST80_1_DM260_EB_Box_User_Data_64_bytes_1[36] := PlcOutputs.ST80_1_DM260_EB_Box_User_Data_64_bytes_1[36];
	HwOutputs.ST80_1_DM260_EB_Box_User_Data_64_bytes_1[37] := PlcOutputs.ST80_1_DM260_EB_Box_User_Data_64_bytes_1[37];
	HwOutputs.ST80_1_DM260_EB_Box_User_Data_64_bytes_1[38] := PlcOutputs.ST80_1_DM260_EB_Box_User_Data_64_bytes_1[38];
	HwOutputs.ST80_1_DM260_EB_Box_User_Data_64_bytes_1[39] := PlcOutputs.ST80_1_DM260_EB_Box_User_Data_64_bytes_1[39];
	HwOutputs.ST80_1_DM260_EB_Box_User_Data_64_bytes_1[40] := PlcOutputs.ST80_1_DM260_EB_Box_User_Data_64_bytes_1[40];
	HwOutputs.ST80_1_DM260_EB_Box_User_Data_64_bytes_1[41] := PlcOutputs.ST80_1_DM260_EB_Box_User_Data_64_bytes_1[41];
	HwOutputs.ST80_1_DM260_EB_Box_User_Data_64_bytes_1[42] := PlcOutputs.ST80_1_DM260_EB_Box_User_Data_64_bytes_1[42];
	HwOutputs.ST80_1_DM260_EB_Box_User_Data_64_bytes_1[43] := PlcOutputs.ST80_1_DM260_EB_Box_User_Data_64_bytes_1[43];
	HwOutputs.ST80_1_DM260_EB_Box_User_Data_64_bytes_1[44] := PlcOutputs.ST80_1_DM260_EB_Box_User_Data_64_bytes_1[44];
	HwOutputs.ST80_1_DM260_EB_Box_User_Data_64_bytes_1[45] := PlcOutputs.ST80_1_DM260_EB_Box_User_Data_64_bytes_1[45];
	HwOutputs.ST80_1_DM260_EB_Box_User_Data_64_bytes_1[46] := PlcOutputs.ST80_1_DM260_EB_Box_User_Data_64_bytes_1[46];
	HwOutputs.ST80_1_DM260_EB_Box_User_Data_64_bytes_1[47] := PlcOutputs.ST80_1_DM260_EB_Box_User_Data_64_bytes_1[47];
	HwOutputs.ST80_1_DM260_EB_Box_User_Data_64_bytes_1[48] := PlcOutputs.ST80_1_DM260_EB_Box_User_Data_64_bytes_1[48];
	HwOutputs.ST80_1_DM260_EB_Box_User_Data_64_bytes_1[49] := PlcOutputs.ST80_1_DM260_EB_Box_User_Data_64_bytes_1[49];
	HwOutputs.ST80_1_DM260_EB_Box_User_Data_64_bytes_1[50] := PlcOutputs.ST80_1_DM260_EB_Box_User_Data_64_bytes_1[50];
	HwOutputs.ST80_1_DM260_EB_Box_User_Data_64_bytes_1[51] := PlcOutputs.ST80_1_DM260_EB_Box_User_Data_64_bytes_1[51];
	HwOutputs.ST80_1_DM260_EB_Box_User_Data_64_bytes_1[52] := PlcOutputs.ST80_1_DM260_EB_Box_User_Data_64_bytes_1[52];
	HwOutputs.ST80_1_DM260_EB_Box_User_Data_64_bytes_1[53] := PlcOutputs.ST80_1_DM260_EB_Box_User_Data_64_bytes_1[53];
	HwOutputs.ST80_1_DM260_EB_Box_User_Data_64_bytes_1[54] := PlcOutputs.ST80_1_DM260_EB_Box_User_Data_64_bytes_1[54];
	HwOutputs.ST80_1_DM260_EB_Box_User_Data_64_bytes_1[55] := PlcOutputs.ST80_1_DM260_EB_Box_User_Data_64_bytes_1[55];
	HwOutputs.ST80_1_DM260_EB_Box_User_Data_64_bytes_1[56] := PlcOutputs.ST80_1_DM260_EB_Box_User_Data_64_bytes_1[56];
	HwOutputs.ST80_1_DM260_EB_Box_User_Data_64_bytes_1[57] := PlcOutputs.ST80_1_DM260_EB_Box_User_Data_64_bytes_1[57];
	HwOutputs.ST80_1_DM260_EB_Box_User_Data_64_bytes_1[58] := PlcOutputs.ST80_1_DM260_EB_Box_User_Data_64_bytes_1[58];
	HwOutputs.ST80_1_DM260_EB_Box_User_Data_64_bytes_1[59] := PlcOutputs.ST80_1_DM260_EB_Box_User_Data_64_bytes_1[59];
	HwOutputs.ST80_1_DM260_EB_Box_User_Data_64_bytes_1[60] := PlcOutputs.ST80_1_DM260_EB_Box_User_Data_64_bytes_1[60];
	HwOutputs.ST80_1_DM260_EB_Box_User_Data_64_bytes_1[61] := PlcOutputs.ST80_1_DM260_EB_Box_User_Data_64_bytes_1[61];
	HwOutputs.ST80_1_DM260_EB_Box_User_Data_64_bytes_1[62] := PlcOutputs.ST80_1_DM260_EB_Box_User_Data_64_bytes_1[62];
	HwOutputs.ST80_1_DM260_EB_Box_User_Data_64_bytes_1[63] := PlcOutputs.ST80_1_DM260_EB_Box_User_Data_64_bytes_1[63];
	HwOutputs.ST80_1_DM260_EB_Box_User_Data_64_bytes_1[64] := PlcOutputs.ST80_1_DM260_EB_Box_User_Data_64_bytes_1[64];
	HwOutputs.ST80_1_DM260_EB_Box_User_Data_64_bytes_1[65] := PlcOutputs.ST80_1_DM260_EB_Box_User_Data_64_bytes_1[65];
	HwOutputs.ST80_1_DM260_EB_Box_User_Data_64_bytes_1[66] := PlcOutputs.ST80_1_DM260_EB_Box_User_Data_64_bytes_1[66];
	HwOutputs.ST80_1_DM260_EB_Box_User_Data_64_bytes_1[67] := PlcOutputs.ST80_1_DM260_EB_Box_User_Data_64_bytes_1[67];
	HwOutputs.ST80_1_DM260_PB_Box_Acquisition_Control_1 := PlcOutputs.ST80_1_DM260_PB_Box_Acquisition_Control_1;
	HwOutputs.ST80_1_DM260_PB_Box_Results_Control_1 := PlcOutputs.ST80_1_DM260_PB_Box_Results_Control_1;
	HwOutputs.ST80_1_DM260_PB_Box_Soft_Event_Control_1 := PlcOutputs.ST80_1_DM260_PB_Box_Soft_Event_Control_1;
	HwOutputs.ST80_1_DM260_PB_Box_User_Data_64_bytes_1[0] := PlcOutputs.ST80_1_DM260_PB_Box_User_Data_64_bytes_1[0];
	HwOutputs.ST80_1_DM260_PB_Box_User_Data_64_bytes_1[1] := PlcOutputs.ST80_1_DM260_PB_Box_User_Data_64_bytes_1[1];
	HwOutputs.ST80_1_DM260_PB_Box_User_Data_64_bytes_1[2] := PlcOutputs.ST80_1_DM260_PB_Box_User_Data_64_bytes_1[2];
	HwOutputs.ST80_1_DM260_PB_Box_User_Data_64_bytes_1[3] := PlcOutputs.ST80_1_DM260_PB_Box_User_Data_64_bytes_1[3];
	HwOutputs.ST80_1_DM260_PB_Box_User_Data_64_bytes_1[4] := PlcOutputs.ST80_1_DM260_PB_Box_User_Data_64_bytes_1[4];
	HwOutputs.ST80_1_DM260_PB_Box_User_Data_64_bytes_1[5] := PlcOutputs.ST80_1_DM260_PB_Box_User_Data_64_bytes_1[5];
	HwOutputs.ST80_1_DM260_PB_Box_User_Data_64_bytes_1[6] := PlcOutputs.ST80_1_DM260_PB_Box_User_Data_64_bytes_1[6];
	HwOutputs.ST80_1_DM260_PB_Box_User_Data_64_bytes_1[7] := PlcOutputs.ST80_1_DM260_PB_Box_User_Data_64_bytes_1[7];
	HwOutputs.ST80_1_DM260_PB_Box_User_Data_64_bytes_1[8] := PlcOutputs.ST80_1_DM260_PB_Box_User_Data_64_bytes_1[8];
	HwOutputs.ST80_1_DM260_PB_Box_User_Data_64_bytes_1[9] := PlcOutputs.ST80_1_DM260_PB_Box_User_Data_64_bytes_1[9];
	HwOutputs.ST80_1_DM260_PB_Box_User_Data_64_bytes_1[10] := PlcOutputs.ST80_1_DM260_PB_Box_User_Data_64_bytes_1[10];
	HwOutputs.ST80_1_DM260_PB_Box_User_Data_64_bytes_1[11] := PlcOutputs.ST80_1_DM260_PB_Box_User_Data_64_bytes_1[11];
	HwOutputs.ST80_1_DM260_PB_Box_User_Data_64_bytes_1[12] := PlcOutputs.ST80_1_DM260_PB_Box_User_Data_64_bytes_1[12];
	HwOutputs.ST80_1_DM260_PB_Box_User_Data_64_bytes_1[13] := PlcOutputs.ST80_1_DM260_PB_Box_User_Data_64_bytes_1[13];
	HwOutputs.ST80_1_DM260_PB_Box_User_Data_64_bytes_1[14] := PlcOutputs.ST80_1_DM260_PB_Box_User_Data_64_bytes_1[14];
	HwOutputs.ST80_1_DM260_PB_Box_User_Data_64_bytes_1[15] := PlcOutputs.ST80_1_DM260_PB_Box_User_Data_64_bytes_1[15];
	HwOutputs.ST80_1_DM260_PB_Box_User_Data_64_bytes_1[16] := PlcOutputs.ST80_1_DM260_PB_Box_User_Data_64_bytes_1[16];
	HwOutputs.ST80_1_DM260_PB_Box_User_Data_64_bytes_1[17] := PlcOutputs.ST80_1_DM260_PB_Box_User_Data_64_bytes_1[17];
	HwOutputs.ST80_1_DM260_PB_Box_User_Data_64_bytes_1[18] := PlcOutputs.ST80_1_DM260_PB_Box_User_Data_64_bytes_1[18];
	HwOutputs.ST80_1_DM260_PB_Box_User_Data_64_bytes_1[19] := PlcOutputs.ST80_1_DM260_PB_Box_User_Data_64_bytes_1[19];
	HwOutputs.ST80_1_DM260_PB_Box_User_Data_64_bytes_1[20] := PlcOutputs.ST80_1_DM260_PB_Box_User_Data_64_bytes_1[20];
	HwOutputs.ST80_1_DM260_PB_Box_User_Data_64_bytes_1[21] := PlcOutputs.ST80_1_DM260_PB_Box_User_Data_64_bytes_1[21];
	HwOutputs.ST80_1_DM260_PB_Box_User_Data_64_bytes_1[22] := PlcOutputs.ST80_1_DM260_PB_Box_User_Data_64_bytes_1[22];
	HwOutputs.ST80_1_DM260_PB_Box_User_Data_64_bytes_1[23] := PlcOutputs.ST80_1_DM260_PB_Box_User_Data_64_bytes_1[23];
	HwOutputs.ST80_1_DM260_PB_Box_User_Data_64_bytes_1[24] := PlcOutputs.ST80_1_DM260_PB_Box_User_Data_64_bytes_1[24];
	HwOutputs.ST80_1_DM260_PB_Box_User_Data_64_bytes_1[25] := PlcOutputs.ST80_1_DM260_PB_Box_User_Data_64_bytes_1[25];
	HwOutputs.ST80_1_DM260_PB_Box_User_Data_64_bytes_1[26] := PlcOutputs.ST80_1_DM260_PB_Box_User_Data_64_bytes_1[26];
	HwOutputs.ST80_1_DM260_PB_Box_User_Data_64_bytes_1[27] := PlcOutputs.ST80_1_DM260_PB_Box_User_Data_64_bytes_1[27];
	HwOutputs.ST80_1_DM260_PB_Box_User_Data_64_bytes_1[28] := PlcOutputs.ST80_1_DM260_PB_Box_User_Data_64_bytes_1[28];
	HwOutputs.ST80_1_DM260_PB_Box_User_Data_64_bytes_1[29] := PlcOutputs.ST80_1_DM260_PB_Box_User_Data_64_bytes_1[29];
	HwOutputs.ST80_1_DM260_PB_Box_User_Data_64_bytes_1[30] := PlcOutputs.ST80_1_DM260_PB_Box_User_Data_64_bytes_1[30];
	HwOutputs.ST80_1_DM260_PB_Box_User_Data_64_bytes_1[31] := PlcOutputs.ST80_1_DM260_PB_Box_User_Data_64_bytes_1[31];
	HwOutputs.ST80_1_DM260_PB_Box_User_Data_64_bytes_1[32] := PlcOutputs.ST80_1_DM260_PB_Box_User_Data_64_bytes_1[32];
	HwOutputs.ST80_1_DM260_PB_Box_User_Data_64_bytes_1[33] := PlcOutputs.ST80_1_DM260_PB_Box_User_Data_64_bytes_1[33];
	HwOutputs.ST80_1_DM260_PB_Box_User_Data_64_bytes_1[34] := PlcOutputs.ST80_1_DM260_PB_Box_User_Data_64_bytes_1[34];
	HwOutputs.ST80_1_DM260_PB_Box_User_Data_64_bytes_1[35] := PlcOutputs.ST80_1_DM260_PB_Box_User_Data_64_bytes_1[35];
	HwOutputs.ST80_1_DM260_PB_Box_User_Data_64_bytes_1[36] := PlcOutputs.ST80_1_DM260_PB_Box_User_Data_64_bytes_1[36];
	HwOutputs.ST80_1_DM260_PB_Box_User_Data_64_bytes_1[37] := PlcOutputs.ST80_1_DM260_PB_Box_User_Data_64_bytes_1[37];
	HwOutputs.ST80_1_DM260_PB_Box_User_Data_64_bytes_1[38] := PlcOutputs.ST80_1_DM260_PB_Box_User_Data_64_bytes_1[38];
	HwOutputs.ST80_1_DM260_PB_Box_User_Data_64_bytes_1[39] := PlcOutputs.ST80_1_DM260_PB_Box_User_Data_64_bytes_1[39];
	HwOutputs.ST80_1_DM260_PB_Box_User_Data_64_bytes_1[40] := PlcOutputs.ST80_1_DM260_PB_Box_User_Data_64_bytes_1[40];
	HwOutputs.ST80_1_DM260_PB_Box_User_Data_64_bytes_1[41] := PlcOutputs.ST80_1_DM260_PB_Box_User_Data_64_bytes_1[41];
	HwOutputs.ST80_1_DM260_PB_Box_User_Data_64_bytes_1[42] := PlcOutputs.ST80_1_DM260_PB_Box_User_Data_64_bytes_1[42];
	HwOutputs.ST80_1_DM260_PB_Box_User_Data_64_bytes_1[43] := PlcOutputs.ST80_1_DM260_PB_Box_User_Data_64_bytes_1[43];
	HwOutputs.ST80_1_DM260_PB_Box_User_Data_64_bytes_1[44] := PlcOutputs.ST80_1_DM260_PB_Box_User_Data_64_bytes_1[44];
	HwOutputs.ST80_1_DM260_PB_Box_User_Data_64_bytes_1[45] := PlcOutputs.ST80_1_DM260_PB_Box_User_Data_64_bytes_1[45];
	HwOutputs.ST80_1_DM260_PB_Box_User_Data_64_bytes_1[46] := PlcOutputs.ST80_1_DM260_PB_Box_User_Data_64_bytes_1[46];
	HwOutputs.ST80_1_DM260_PB_Box_User_Data_64_bytes_1[47] := PlcOutputs.ST80_1_DM260_PB_Box_User_Data_64_bytes_1[47];
	HwOutputs.ST80_1_DM260_PB_Box_User_Data_64_bytes_1[48] := PlcOutputs.ST80_1_DM260_PB_Box_User_Data_64_bytes_1[48];
	HwOutputs.ST80_1_DM260_PB_Box_User_Data_64_bytes_1[49] := PlcOutputs.ST80_1_DM260_PB_Box_User_Data_64_bytes_1[49];
	HwOutputs.ST80_1_DM260_PB_Box_User_Data_64_bytes_1[50] := PlcOutputs.ST80_1_DM260_PB_Box_User_Data_64_bytes_1[50];
	HwOutputs.ST80_1_DM260_PB_Box_User_Data_64_bytes_1[51] := PlcOutputs.ST80_1_DM260_PB_Box_User_Data_64_bytes_1[51];
	HwOutputs.ST80_1_DM260_PB_Box_User_Data_64_bytes_1[52] := PlcOutputs.ST80_1_DM260_PB_Box_User_Data_64_bytes_1[52];
	HwOutputs.ST80_1_DM260_PB_Box_User_Data_64_bytes_1[53] := PlcOutputs.ST80_1_DM260_PB_Box_User_Data_64_bytes_1[53];
	HwOutputs.ST80_1_DM260_PB_Box_User_Data_64_bytes_1[54] := PlcOutputs.ST80_1_DM260_PB_Box_User_Data_64_bytes_1[54];
	HwOutputs.ST80_1_DM260_PB_Box_User_Data_64_bytes_1[55] := PlcOutputs.ST80_1_DM260_PB_Box_User_Data_64_bytes_1[55];
	HwOutputs.ST80_1_DM260_PB_Box_User_Data_64_bytes_1[56] := PlcOutputs.ST80_1_DM260_PB_Box_User_Data_64_bytes_1[56];
	HwOutputs.ST80_1_DM260_PB_Box_User_Data_64_bytes_1[57] := PlcOutputs.ST80_1_DM260_PB_Box_User_Data_64_bytes_1[57];
	HwOutputs.ST80_1_DM260_PB_Box_User_Data_64_bytes_1[58] := PlcOutputs.ST80_1_DM260_PB_Box_User_Data_64_bytes_1[58];
	HwOutputs.ST80_1_DM260_PB_Box_User_Data_64_bytes_1[59] := PlcOutputs.ST80_1_DM260_PB_Box_User_Data_64_bytes_1[59];
	HwOutputs.ST80_1_DM260_PB_Box_User_Data_64_bytes_1[60] := PlcOutputs.ST80_1_DM260_PB_Box_User_Data_64_bytes_1[60];
	HwOutputs.ST80_1_DM260_PB_Box_User_Data_64_bytes_1[61] := PlcOutputs.ST80_1_DM260_PB_Box_User_Data_64_bytes_1[61];
	HwOutputs.ST80_1_DM260_PB_Box_User_Data_64_bytes_1[62] := PlcOutputs.ST80_1_DM260_PB_Box_User_Data_64_bytes_1[62];
	HwOutputs.ST80_1_DM260_PB_Box_User_Data_64_bytes_1[63] := PlcOutputs.ST80_1_DM260_PB_Box_User_Data_64_bytes_1[63];
	HwOutputs.ST80_1_DM260_PB_Box_User_Data_64_bytes_1[64] := PlcOutputs.ST80_1_DM260_PB_Box_User_Data_64_bytes_1[64];
	HwOutputs.ST80_1_DM260_PB_Box_User_Data_64_bytes_1[65] := PlcOutputs.ST80_1_DM260_PB_Box_User_Data_64_bytes_1[65];
	HwOutputs.ST80_1_DM260_PB_Box_User_Data_64_bytes_1[66] := PlcOutputs.ST80_1_DM260_PB_Box_User_Data_64_bytes_1[66];
	HwOutputs.ST80_1_DM260_PB_Box_User_Data_64_bytes_1[67] := PlcOutputs.ST80_1_DM260_PB_Box_User_Data_64_bytes_1[67];
	HwOutputs.ST80_ET200SP_2_11M1 := PlcOutputs.ST80_ET200SP_2_11M1;
	HwOutputs.ST80_ET200SP_2_11M2 := PlcOutputs.ST80_ET200SP_2_11M2;
	HwOutputs.ST80_ET200SP_2_11M3 := PlcOutputs.ST80_ET200SP_2_11M3;
	HwOutputs.ST80_ET200SP_2_11M4 := PlcOutputs.ST80_ET200SP_2_11M4;
	HwOutputs.ST80_ET200SP_2_12M1 := PlcOutputs.ST80_ET200SP_2_12M1;
	HwOutputs.ST80_ET200SP_2_12M2 := PlcOutputs.ST80_ET200SP_2_12M2;
	HwOutputs.ST80_ET200SP_2_12M3 := PlcOutputs.ST80_ET200SP_2_12M3;
	HwOutputs.ST80_ET200SP_2_12M4 := PlcOutputs.ST80_ET200SP_2_12M4;
	HwOutputs.ST80_ET200SP_2_13M1 := PlcOutputs.ST80_ET200SP_2_13M1;
	HwOutputs.ST80_ET200SP_2_13M2 := PlcOutputs.ST80_ET200SP_2_13M2;
	HwOutputs.ST80_ET200SP_2_13M3 := PlcOutputs.ST80_ET200SP_2_13M3;
	HwOutputs.ST80_ET200SP_2_13M4 := PlcOutputs.ST80_ET200SP_2_13M4;
	HwOutputs.ST80_1_TZ535_PN_In_Out_32_byte_1[0] := PlcOutputs.ST80_1_TZ535_PN_In_Out_32_byte_1[0];
	HwOutputs.ST80_1_TZ535_PN_In_Out_32_byte_1[1] := PlcOutputs.ST80_1_TZ535_PN_In_Out_32_byte_1[1];
	HwOutputs.ST80_1_TZ535_PN_In_Out_32_byte_1[2] := PlcOutputs.ST80_1_TZ535_PN_In_Out_32_byte_1[2];
	HwOutputs.ST80_1_TZ535_PN_In_Out_32_byte_1[3] := PlcOutputs.ST80_1_TZ535_PN_In_Out_32_byte_1[3];
	HwOutputs.ST80_1_TZ535_PN_In_Out_32_byte_1[4] := PlcOutputs.ST80_1_TZ535_PN_In_Out_32_byte_1[4];
	HwOutputs.ST80_1_TZ535_PN_In_Out_32_byte_1[5] := PlcOutputs.ST80_1_TZ535_PN_In_Out_32_byte_1[5];
	HwOutputs.ST80_1_TZ535_PN_In_Out_32_byte_1[6] := PlcOutputs.ST80_1_TZ535_PN_In_Out_32_byte_1[6];
	HwOutputs.ST80_1_TZ535_PN_In_Out_32_byte_1[7] := PlcOutputs.ST80_1_TZ535_PN_In_Out_32_byte_1[7];
	HwOutputs.ST80_1_TZ535_PN_In_Out_32_byte_1[8] := PlcOutputs.ST80_1_TZ535_PN_In_Out_32_byte_1[8];
	HwOutputs.ST80_1_TZ535_PN_In_Out_32_byte_1[9] := PlcOutputs.ST80_1_TZ535_PN_In_Out_32_byte_1[9];
	HwOutputs.ST80_1_TZ535_PN_In_Out_32_byte_1[10] := PlcOutputs.ST80_1_TZ535_PN_In_Out_32_byte_1[10];
	HwOutputs.ST80_1_TZ535_PN_In_Out_32_byte_1[11] := PlcOutputs.ST80_1_TZ535_PN_In_Out_32_byte_1[11];
	HwOutputs.ST80_1_TZ535_PN_In_Out_32_byte_1[12] := PlcOutputs.ST80_1_TZ535_PN_In_Out_32_byte_1[12];
	HwOutputs.ST80_1_TZ535_PN_In_Out_32_byte_1[13] := PlcOutputs.ST80_1_TZ535_PN_In_Out_32_byte_1[13];
	HwOutputs.ST80_1_TZ535_PN_In_Out_32_byte_1[14] := PlcOutputs.ST80_1_TZ535_PN_In_Out_32_byte_1[14];
	HwOutputs.ST80_1_TZ535_PN_In_Out_32_byte_1[15] := PlcOutputs.ST80_1_TZ535_PN_In_Out_32_byte_1[15];
	HwOutputs.ST80_1_TZ535_PN_In_Out_32_byte_1[16] := PlcOutputs.ST80_1_TZ535_PN_In_Out_32_byte_1[16];
	HwOutputs.ST80_1_TZ535_PN_In_Out_32_byte_1[17] := PlcOutputs.ST80_1_TZ535_PN_In_Out_32_byte_1[17];
	HwOutputs.ST80_1_TZ535_PN_In_Out_32_byte_1[18] := PlcOutputs.ST80_1_TZ535_PN_In_Out_32_byte_1[18];
	HwOutputs.ST80_1_TZ535_PN_In_Out_32_byte_1[19] := PlcOutputs.ST80_1_TZ535_PN_In_Out_32_byte_1[19];
	HwOutputs.ST80_1_TZ535_PN_In_Out_32_byte_1[20] := PlcOutputs.ST80_1_TZ535_PN_In_Out_32_byte_1[20];
	HwOutputs.ST80_1_TZ535_PN_In_Out_32_byte_1[21] := PlcOutputs.ST80_1_TZ535_PN_In_Out_32_byte_1[21];
	HwOutputs.ST80_1_TZ535_PN_In_Out_32_byte_1[22] := PlcOutputs.ST80_1_TZ535_PN_In_Out_32_byte_1[22];
	HwOutputs.ST80_1_TZ535_PN_In_Out_32_byte_1[23] := PlcOutputs.ST80_1_TZ535_PN_In_Out_32_byte_1[23];
	HwOutputs.ST80_1_TZ535_PN_In_Out_32_byte_1[24] := PlcOutputs.ST80_1_TZ535_PN_In_Out_32_byte_1[24];
	HwOutputs.ST80_1_TZ535_PN_In_Out_32_byte_1[25] := PlcOutputs.ST80_1_TZ535_PN_In_Out_32_byte_1[25];
	HwOutputs.ST80_1_TZ535_PN_In_Out_32_byte_1[26] := PlcOutputs.ST80_1_TZ535_PN_In_Out_32_byte_1[26];
	HwOutputs.ST80_1_TZ535_PN_In_Out_32_byte_1[27] := PlcOutputs.ST80_1_TZ535_PN_In_Out_32_byte_1[27];
	HwOutputs.ST80_1_TZ535_PN_In_Out_32_byte_1[28] := PlcOutputs.ST80_1_TZ535_PN_In_Out_32_byte_1[28];
	HwOutputs.ST80_1_TZ535_PN_In_Out_32_byte_1[29] := PlcOutputs.ST80_1_TZ535_PN_In_Out_32_byte_1[29];
	HwOutputs.ST80_1_TZ535_PN_In_Out_32_byte_1[30] := PlcOutputs.ST80_1_TZ535_PN_In_Out_32_byte_1[30];
	HwOutputs.ST80_1_TZ535_PN_In_Out_32_byte_1[31] := PlcOutputs.ST80_1_TZ535_PN_In_Out_32_byte_1[31];
	HwOutputs.ST80_1_DM260_Housing_Acquisition_Control_1 := PlcOutputs.ST80_1_DM260_Housing_Acquisition_Control_1;
	HwOutputs.ST80_1_DM260_Housing_Results_Control_1 := PlcOutputs.ST80_1_DM260_Housing_Results_Control_1;
	HwOutputs.ST80_1_DM260_Housing_Soft_Event_Control_1 := PlcOutputs.ST80_1_DM260_Housing_Soft_Event_Control_1;
	HwOutputs.ST80_1_DM260_Housing_User_Data_64_bytes_1[0] := PlcOutputs.ST80_1_DM260_Housing_User_Data_64_bytes_1[0];
	HwOutputs.ST80_1_DM260_Housing_User_Data_64_bytes_1[1] := PlcOutputs.ST80_1_DM260_Housing_User_Data_64_bytes_1[1];
	HwOutputs.ST80_1_DM260_Housing_User_Data_64_bytes_1[2] := PlcOutputs.ST80_1_DM260_Housing_User_Data_64_bytes_1[2];
	HwOutputs.ST80_1_DM260_Housing_User_Data_64_bytes_1[3] := PlcOutputs.ST80_1_DM260_Housing_User_Data_64_bytes_1[3];
	HwOutputs.ST80_1_DM260_Housing_User_Data_64_bytes_1[4] := PlcOutputs.ST80_1_DM260_Housing_User_Data_64_bytes_1[4];
	HwOutputs.ST80_1_DM260_Housing_User_Data_64_bytes_1[5] := PlcOutputs.ST80_1_DM260_Housing_User_Data_64_bytes_1[5];
	HwOutputs.ST80_1_DM260_Housing_User_Data_64_bytes_1[6] := PlcOutputs.ST80_1_DM260_Housing_User_Data_64_bytes_1[6];
	HwOutputs.ST80_1_DM260_Housing_User_Data_64_bytes_1[7] := PlcOutputs.ST80_1_DM260_Housing_User_Data_64_bytes_1[7];
	HwOutputs.ST80_1_DM260_Housing_User_Data_64_bytes_1[8] := PlcOutputs.ST80_1_DM260_Housing_User_Data_64_bytes_1[8];
	HwOutputs.ST80_1_DM260_Housing_User_Data_64_bytes_1[9] := PlcOutputs.ST80_1_DM260_Housing_User_Data_64_bytes_1[9];
	HwOutputs.ST80_1_DM260_Housing_User_Data_64_bytes_1[10] := PlcOutputs.ST80_1_DM260_Housing_User_Data_64_bytes_1[10];
	HwOutputs.ST80_1_DM260_Housing_User_Data_64_bytes_1[11] := PlcOutputs.ST80_1_DM260_Housing_User_Data_64_bytes_1[11];
	HwOutputs.ST80_1_DM260_Housing_User_Data_64_bytes_1[12] := PlcOutputs.ST80_1_DM260_Housing_User_Data_64_bytes_1[12];
	HwOutputs.ST80_1_DM260_Housing_User_Data_64_bytes_1[13] := PlcOutputs.ST80_1_DM260_Housing_User_Data_64_bytes_1[13];
	HwOutputs.ST80_1_DM260_Housing_User_Data_64_bytes_1[14] := PlcOutputs.ST80_1_DM260_Housing_User_Data_64_bytes_1[14];
	HwOutputs.ST80_1_DM260_Housing_User_Data_64_bytes_1[15] := PlcOutputs.ST80_1_DM260_Housing_User_Data_64_bytes_1[15];
	HwOutputs.ST80_1_DM260_Housing_User_Data_64_bytes_1[16] := PlcOutputs.ST80_1_DM260_Housing_User_Data_64_bytes_1[16];
	HwOutputs.ST80_1_DM260_Housing_User_Data_64_bytes_1[17] := PlcOutputs.ST80_1_DM260_Housing_User_Data_64_bytes_1[17];
	HwOutputs.ST80_1_DM260_Housing_User_Data_64_bytes_1[18] := PlcOutputs.ST80_1_DM260_Housing_User_Data_64_bytes_1[18];
	HwOutputs.ST80_1_DM260_Housing_User_Data_64_bytes_1[19] := PlcOutputs.ST80_1_DM260_Housing_User_Data_64_bytes_1[19];
	HwOutputs.ST80_1_DM260_Housing_User_Data_64_bytes_1[20] := PlcOutputs.ST80_1_DM260_Housing_User_Data_64_bytes_1[20];
	HwOutputs.ST80_1_DM260_Housing_User_Data_64_bytes_1[21] := PlcOutputs.ST80_1_DM260_Housing_User_Data_64_bytes_1[21];
	HwOutputs.ST80_1_DM260_Housing_User_Data_64_bytes_1[22] := PlcOutputs.ST80_1_DM260_Housing_User_Data_64_bytes_1[22];
	HwOutputs.ST80_1_DM260_Housing_User_Data_64_bytes_1[23] := PlcOutputs.ST80_1_DM260_Housing_User_Data_64_bytes_1[23];
	HwOutputs.ST80_1_DM260_Housing_User_Data_64_bytes_1[24] := PlcOutputs.ST80_1_DM260_Housing_User_Data_64_bytes_1[24];
	HwOutputs.ST80_1_DM260_Housing_User_Data_64_bytes_1[25] := PlcOutputs.ST80_1_DM260_Housing_User_Data_64_bytes_1[25];
	HwOutputs.ST80_1_DM260_Housing_User_Data_64_bytes_1[26] := PlcOutputs.ST80_1_DM260_Housing_User_Data_64_bytes_1[26];
	HwOutputs.ST80_1_DM260_Housing_User_Data_64_bytes_1[27] := PlcOutputs.ST80_1_DM260_Housing_User_Data_64_bytes_1[27];
	HwOutputs.ST80_1_DM260_Housing_User_Data_64_bytes_1[28] := PlcOutputs.ST80_1_DM260_Housing_User_Data_64_bytes_1[28];
	HwOutputs.ST80_1_DM260_Housing_User_Data_64_bytes_1[29] := PlcOutputs.ST80_1_DM260_Housing_User_Data_64_bytes_1[29];
	HwOutputs.ST80_1_DM260_Housing_User_Data_64_bytes_1[30] := PlcOutputs.ST80_1_DM260_Housing_User_Data_64_bytes_1[30];
	HwOutputs.ST80_1_DM260_Housing_User_Data_64_bytes_1[31] := PlcOutputs.ST80_1_DM260_Housing_User_Data_64_bytes_1[31];
	HwOutputs.ST80_1_DM260_Housing_User_Data_64_bytes_1[32] := PlcOutputs.ST80_1_DM260_Housing_User_Data_64_bytes_1[32];
	HwOutputs.ST80_1_DM260_Housing_User_Data_64_bytes_1[33] := PlcOutputs.ST80_1_DM260_Housing_User_Data_64_bytes_1[33];
	HwOutputs.ST80_1_DM260_Housing_User_Data_64_bytes_1[34] := PlcOutputs.ST80_1_DM260_Housing_User_Data_64_bytes_1[34];
	HwOutputs.ST80_1_DM260_Housing_User_Data_64_bytes_1[35] := PlcOutputs.ST80_1_DM260_Housing_User_Data_64_bytes_1[35];
	HwOutputs.ST80_1_DM260_Housing_User_Data_64_bytes_1[36] := PlcOutputs.ST80_1_DM260_Housing_User_Data_64_bytes_1[36];
	HwOutputs.ST80_1_DM260_Housing_User_Data_64_bytes_1[37] := PlcOutputs.ST80_1_DM260_Housing_User_Data_64_bytes_1[37];
	HwOutputs.ST80_1_DM260_Housing_User_Data_64_bytes_1[38] := PlcOutputs.ST80_1_DM260_Housing_User_Data_64_bytes_1[38];
	HwOutputs.ST80_1_DM260_Housing_User_Data_64_bytes_1[39] := PlcOutputs.ST80_1_DM260_Housing_User_Data_64_bytes_1[39];
	HwOutputs.ST80_1_DM260_Housing_User_Data_64_bytes_1[40] := PlcOutputs.ST80_1_DM260_Housing_User_Data_64_bytes_1[40];
	HwOutputs.ST80_1_DM260_Housing_User_Data_64_bytes_1[41] := PlcOutputs.ST80_1_DM260_Housing_User_Data_64_bytes_1[41];
	HwOutputs.ST80_1_DM260_Housing_User_Data_64_bytes_1[42] := PlcOutputs.ST80_1_DM260_Housing_User_Data_64_bytes_1[42];
	HwOutputs.ST80_1_DM260_Housing_User_Data_64_bytes_1[43] := PlcOutputs.ST80_1_DM260_Housing_User_Data_64_bytes_1[43];
	HwOutputs.ST80_1_DM260_Housing_User_Data_64_bytes_1[44] := PlcOutputs.ST80_1_DM260_Housing_User_Data_64_bytes_1[44];
	HwOutputs.ST80_1_DM260_Housing_User_Data_64_bytes_1[45] := PlcOutputs.ST80_1_DM260_Housing_User_Data_64_bytes_1[45];
	HwOutputs.ST80_1_DM260_Housing_User_Data_64_bytes_1[46] := PlcOutputs.ST80_1_DM260_Housing_User_Data_64_bytes_1[46];
	HwOutputs.ST80_1_DM260_Housing_User_Data_64_bytes_1[47] := PlcOutputs.ST80_1_DM260_Housing_User_Data_64_bytes_1[47];
	HwOutputs.ST80_1_DM260_Housing_User_Data_64_bytes_1[48] := PlcOutputs.ST80_1_DM260_Housing_User_Data_64_bytes_1[48];
	HwOutputs.ST80_1_DM260_Housing_User_Data_64_bytes_1[49] := PlcOutputs.ST80_1_DM260_Housing_User_Data_64_bytes_1[49];
	HwOutputs.ST80_1_DM260_Housing_User_Data_64_bytes_1[50] := PlcOutputs.ST80_1_DM260_Housing_User_Data_64_bytes_1[50];
	HwOutputs.ST80_1_DM260_Housing_User_Data_64_bytes_1[51] := PlcOutputs.ST80_1_DM260_Housing_User_Data_64_bytes_1[51];
	HwOutputs.ST80_1_DM260_Housing_User_Data_64_bytes_1[52] := PlcOutputs.ST80_1_DM260_Housing_User_Data_64_bytes_1[52];
	HwOutputs.ST80_1_DM260_Housing_User_Data_64_bytes_1[53] := PlcOutputs.ST80_1_DM260_Housing_User_Data_64_bytes_1[53];
	HwOutputs.ST80_1_DM260_Housing_User_Data_64_bytes_1[54] := PlcOutputs.ST80_1_DM260_Housing_User_Data_64_bytes_1[54];
	HwOutputs.ST80_1_DM260_Housing_User_Data_64_bytes_1[55] := PlcOutputs.ST80_1_DM260_Housing_User_Data_64_bytes_1[55];
	HwOutputs.ST80_1_DM260_Housing_User_Data_64_bytes_1[56] := PlcOutputs.ST80_1_DM260_Housing_User_Data_64_bytes_1[56];
	HwOutputs.ST80_1_DM260_Housing_User_Data_64_bytes_1[57] := PlcOutputs.ST80_1_DM260_Housing_User_Data_64_bytes_1[57];
	HwOutputs.ST80_1_DM260_Housing_User_Data_64_bytes_1[58] := PlcOutputs.ST80_1_DM260_Housing_User_Data_64_bytes_1[58];
	HwOutputs.ST80_1_DM260_Housing_User_Data_64_bytes_1[59] := PlcOutputs.ST80_1_DM260_Housing_User_Data_64_bytes_1[59];
	HwOutputs.ST80_1_DM260_Housing_User_Data_64_bytes_1[60] := PlcOutputs.ST80_1_DM260_Housing_User_Data_64_bytes_1[60];
	HwOutputs.ST80_1_DM260_Housing_User_Data_64_bytes_1[61] := PlcOutputs.ST80_1_DM260_Housing_User_Data_64_bytes_1[61];
	HwOutputs.ST80_1_DM260_Housing_User_Data_64_bytes_1[62] := PlcOutputs.ST80_1_DM260_Housing_User_Data_64_bytes_1[62];
	HwOutputs.ST80_1_DM260_Housing_User_Data_64_bytes_1[63] := PlcOutputs.ST80_1_DM260_Housing_User_Data_64_bytes_1[63];
	HwOutputs.ST80_1_DM260_Housing_User_Data_64_bytes_1[64] := PlcOutputs.ST80_1_DM260_Housing_User_Data_64_bytes_1[64];
	HwOutputs.ST80_1_DM260_Housing_User_Data_64_bytes_1[65] := PlcOutputs.ST80_1_DM260_Housing_User_Data_64_bytes_1[65];
	HwOutputs.ST80_1_DM260_Housing_User_Data_64_bytes_1[66] := PlcOutputs.ST80_1_DM260_Housing_User_Data_64_bytes_1[66];
	HwOutputs.ST80_1_DM260_Housing_User_Data_64_bytes_1[67] := PlcOutputs.ST80_1_DM260_Housing_User_Data_64_bytes_1[67];
	HwOutputs.ST80_CPX_MPA1S_VMPA1_FB_EMS_8_8DO_1 := PlcOutputs.ST80_CPX_MPA1S_VMPA1_FB_EMS_8_8DO_1;
	HwOutputs.ST80_CPX_MPA1S_VMPA1_FB_EMS_8_8DO_2 := PlcOutputs.ST80_CPX_MPA1S_VMPA1_FB_EMS_8_8DO_2;
	HwOutputs.ST80_CPX_MPA2S_VMPA2_FB_EMS_4_4DO_1 := PlcOutputs.ST80_CPX_MPA2S_VMPA2_FB_EMS_4_4DO_1;
	HwOutputs.ST80_CPX_MPA1S_VMPA1_FB_EMS_8_8DO_3 := PlcOutputs.ST80_CPX_MPA1S_VMPA1_FB_EMS_8_8DO_3;
	HwOutputs.ST80_CPX_MPA2S_VMPA2_FB_EMS_4_4DO_2 := PlcOutputs.ST80_CPX_MPA2S_VMPA2_FB_EMS_4_4DO_2;
	HwOutputs.ST80_CPX_MPA1S_VMPA1_FB_EMS_8_8DO_4 := PlcOutputs.ST80_CPX_MPA1S_VMPA1_FB_EMS_8_8DO_4;
	HwOutputs.ST80_CPX_MPA1S_VMPA1_FB_EMS_8_8DO_5 := PlcOutputs.ST80_CPX_MPA1S_VMPA1_FB_EMS_8_8DO_5;
	HwOutputs.ST80_CPX_MPA1G_VMPA1_FB_EMG_8_8DO_1 := PlcOutputs.ST80_CPX_MPA1G_VMPA1_FB_EMG_8_8DO_1;
	HwOutputs.ST80_CPX_MPA1G_VMPA1_FB_EMG_8_8DO_2 := PlcOutputs.ST80_CPX_MPA1G_VMPA1_FB_EMG_8_8DO_2;
	HwOutputs.ST80_CPX_MPA2G_VMPA2_FB_EMG_4_4DO_1 := PlcOutputs.ST80_CPX_MPA2G_VMPA2_FB_EMG_4_4DO_1;
	HwOutputs.ST80_CPX_MPA1G_VMPA1_FB_EMG_8_8DO_3 := PlcOutputs.ST80_CPX_MPA1G_VMPA1_FB_EMG_8_8DO_3;
	HwOutputs.ST80_CPX_MPA1G_VMPA1_FB_EMG_8_8DO_4 := PlcOutputs.ST80_CPX_MPA1G_VMPA1_FB_EMG_8_8DO_4;
	HwOutputs.ST80_CPX_MPA1G_VMPA1_FB_EMG_8_8DO_5 := PlcOutputs.ST80_CPX_MPA1G_VMPA1_FB_EMG_8_8DO_5;
	HwOutputs.ST80_CPX_MPA1G_VMPA1_FB_EMG_8_8DO_6 := PlcOutputs.ST80_CPX_MPA1G_VMPA1_FB_EMG_8_8DO_6;
	HwOutputs.ST80_ET200SP_CM_4xIO_Link_1[0] := PlcOutputs.ST80_ET200SP_CM_4xIO_Link_1[0];
	HwOutputs.ST80_ET200SP_CM_4xIO_Link_1[1] := PlcOutputs.ST80_ET200SP_CM_4xIO_Link_1[1];
	HwOutputs.ST80_ET200SP_CM_4xIO_Link_1[2] := PlcOutputs.ST80_ET200SP_CM_4xIO_Link_1[2];
	HwOutputs.ST80_ET200SP_CM_4xIO_Link_1[3] := PlcOutputs.ST80_ET200SP_CM_4xIO_Link_1[3];
	HwOutputs.ST80_ET200SP_CM_4xIO_Link_1[4] := PlcOutputs.ST80_ET200SP_CM_4xIO_Link_1[4];
	HwOutputs.ST80_ET200SP_CM_4xIO_Link_1[5] := PlcOutputs.ST80_ET200SP_CM_4xIO_Link_1[5];
	HwOutputs.ST80_ET200SP_CM_4xIO_Link_1[6] := PlcOutputs.ST80_ET200SP_CM_4xIO_Link_1[6];
	HwOutputs.ST80_ET200SP_CM_4xIO_Link_1[7] := PlcOutputs.ST80_ET200SP_CM_4xIO_Link_1[7];
	HwOutputs.ST80_ET200SP_CM_4xIO_Link_1[8] := PlcOutputs.ST80_ET200SP_CM_4xIO_Link_1[8];
	HwOutputs.ST80_ET200SP_CM_4xIO_Link_1[9] := PlcOutputs.ST80_ET200SP_CM_4xIO_Link_1[9];
	HwOutputs.ST80_ET200SP_CM_4xIO_Link_1[10] := PlcOutputs.ST80_ET200SP_CM_4xIO_Link_1[10];
	HwOutputs.ST80_ET200SP_CM_4xIO_Link_1[11] := PlcOutputs.ST80_ET200SP_CM_4xIO_Link_1[11];
	HwOutputs.ST80_ET200SP_CM_4xIO_Link_1[12] := PlcOutputs.ST80_ET200SP_CM_4xIO_Link_1[12];
	HwOutputs.ST80_ET200SP_CM_4xIO_Link_1[13] := PlcOutputs.ST80_ET200SP_CM_4xIO_Link_1[13];
	HwOutputs.ST80_ET200SP_CM_4xIO_Link_1[14] := PlcOutputs.ST80_ET200SP_CM_4xIO_Link_1[14];
	HwOutputs.ST80_ET200SP_CM_4xIO_Link_1[15] := PlcOutputs.ST80_ET200SP_CM_4xIO_Link_1[15];
	HwOutputs.ST80_ET200SP_CM_4xIO_Link_1[16] := PlcOutputs.ST80_ET200SP_CM_4xIO_Link_1[16];
	HwOutputs.ST80_ET200SP_CM_4xIO_Link_1[17] := PlcOutputs.ST80_ET200SP_CM_4xIO_Link_1[17];
	HwOutputs.ST80_ET200SP_CM_4xIO_Link_1[18] := PlcOutputs.ST80_ET200SP_CM_4xIO_Link_1[18];
	HwOutputs.ST80_ET200SP_CM_4xIO_Link_1[19] := PlcOutputs.ST80_ET200SP_CM_4xIO_Link_1[19];
	HwOutputs.ST80_ET200SP_CM_4xIO_Link_1[20] := PlcOutputs.ST80_ET200SP_CM_4xIO_Link_1[20];
	HwOutputs.ST80_ET200SP_CM_4xIO_Link_1[21] := PlcOutputs.ST80_ET200SP_CM_4xIO_Link_1[21];
	HwOutputs.ST80_ET200SP_CM_4xIO_Link_1[22] := PlcOutputs.ST80_ET200SP_CM_4xIO_Link_1[22];
	HwOutputs.ST80_ET200SP_CM_4xIO_Link_1[23] := PlcOutputs.ST80_ET200SP_CM_4xIO_Link_1[23];
	HwOutputs.ST80_ET200SP_CM_4xIO_Link_1[24] := PlcOutputs.ST80_ET200SP_CM_4xIO_Link_1[24];
	HwOutputs.ST80_ET200SP_CM_4xIO_Link_1[25] := PlcOutputs.ST80_ET200SP_CM_4xIO_Link_1[25];
	HwOutputs.ST80_ET200SP_CM_4xIO_Link_1[26] := PlcOutputs.ST80_ET200SP_CM_4xIO_Link_1[26];
	HwOutputs.ST80_ET200SP_CM_4xIO_Link_1[27] := PlcOutputs.ST80_ET200SP_CM_4xIO_Link_1[27];
	HwOutputs.ST80_ET200SP_CM_4xIO_Link_1[28] := PlcOutputs.ST80_ET200SP_CM_4xIO_Link_1[28];
	HwOutputs.ST80_ET200SP_CM_4xIO_Link_1[29] := PlcOutputs.ST80_ET200SP_CM_4xIO_Link_1[29];
	HwOutputs.ST80_ET200SP_CM_4xIO_Link_1[30] := PlcOutputs.ST80_ET200SP_CM_4xIO_Link_1[30];
	HwOutputs.ST80_ET200SP_CM_4xIO_Link_1[31] := PlcOutputs.ST80_ET200SP_CM_4xIO_Link_1[31];
	HwOutputs.ST80_ET200SP_CM_4xIO_Link_2[0] := PlcOutputs.ST80_ET200SP_CM_4xIO_Link_2[0];
	HwOutputs.ST80_ET200SP_CM_4xIO_Link_2[1] := PlcOutputs.ST80_ET200SP_CM_4xIO_Link_2[1];
	HwOutputs.ST80_ET200SP_CM_4xIO_Link_2[2] := PlcOutputs.ST80_ET200SP_CM_4xIO_Link_2[2];
	HwOutputs.ST80_ET200SP_CM_4xIO_Link_2[3] := PlcOutputs.ST80_ET200SP_CM_4xIO_Link_2[3];
	HwOutputs.ST80_ET200SP_CM_4xIO_Link_2[4] := PlcOutputs.ST80_ET200SP_CM_4xIO_Link_2[4];
	HwOutputs.ST80_ET200SP_CM_4xIO_Link_2[5] := PlcOutputs.ST80_ET200SP_CM_4xIO_Link_2[5];
	HwOutputs.ST80_ET200SP_CM_4xIO_Link_2[6] := PlcOutputs.ST80_ET200SP_CM_4xIO_Link_2[6];
	HwOutputs.ST80_ET200SP_CM_4xIO_Link_2[7] := PlcOutputs.ST80_ET200SP_CM_4xIO_Link_2[7];
	HwOutputs.ST80_ET200SP_CM_4xIO_Link_2[8] := PlcOutputs.ST80_ET200SP_CM_4xIO_Link_2[8];
	HwOutputs.ST80_ET200SP_CM_4xIO_Link_2[9] := PlcOutputs.ST80_ET200SP_CM_4xIO_Link_2[9];
	HwOutputs.ST80_ET200SP_CM_4xIO_Link_2[10] := PlcOutputs.ST80_ET200SP_CM_4xIO_Link_2[10];
	HwOutputs.ST80_ET200SP_CM_4xIO_Link_2[11] := PlcOutputs.ST80_ET200SP_CM_4xIO_Link_2[11];
	HwOutputs.ST80_ET200SP_CM_4xIO_Link_2[12] := PlcOutputs.ST80_ET200SP_CM_4xIO_Link_2[12];
	HwOutputs.ST80_ET200SP_CM_4xIO_Link_2[13] := PlcOutputs.ST80_ET200SP_CM_4xIO_Link_2[13];
	HwOutputs.ST80_ET200SP_CM_4xIO_Link_2[14] := PlcOutputs.ST80_ET200SP_CM_4xIO_Link_2[14];
	HwOutputs.ST80_ET200SP_CM_4xIO_Link_2[15] := PlcOutputs.ST80_ET200SP_CM_4xIO_Link_2[15];
	HwOutputs.ST80_ET200SP_CM_4xIO_Link_2[16] := PlcOutputs.ST80_ET200SP_CM_4xIO_Link_2[16];
	HwOutputs.ST80_ET200SP_CM_4xIO_Link_2[17] := PlcOutputs.ST80_ET200SP_CM_4xIO_Link_2[17];
	HwOutputs.ST80_ET200SP_CM_4xIO_Link_2[18] := PlcOutputs.ST80_ET200SP_CM_4xIO_Link_2[18];
	HwOutputs.ST80_ET200SP_CM_4xIO_Link_2[19] := PlcOutputs.ST80_ET200SP_CM_4xIO_Link_2[19];
	HwOutputs.ST80_ET200SP_CM_4xIO_Link_2[20] := PlcOutputs.ST80_ET200SP_CM_4xIO_Link_2[20];
	HwOutputs.ST80_ET200SP_CM_4xIO_Link_2[21] := PlcOutputs.ST80_ET200SP_CM_4xIO_Link_2[21];
	HwOutputs.ST80_ET200SP_CM_4xIO_Link_2[22] := PlcOutputs.ST80_ET200SP_CM_4xIO_Link_2[22];
	HwOutputs.ST80_ET200SP_CM_4xIO_Link_2[23] := PlcOutputs.ST80_ET200SP_CM_4xIO_Link_2[23];
	HwOutputs.ST80_ET200SP_CM_4xIO_Link_2[24] := PlcOutputs.ST80_ET200SP_CM_4xIO_Link_2[24];
	HwOutputs.ST80_ET200SP_CM_4xIO_Link_2[25] := PlcOutputs.ST80_ET200SP_CM_4xIO_Link_2[25];
	HwOutputs.ST80_ET200SP_CM_4xIO_Link_2[26] := PlcOutputs.ST80_ET200SP_CM_4xIO_Link_2[26];
	HwOutputs.ST80_ET200SP_CM_4xIO_Link_2[27] := PlcOutputs.ST80_ET200SP_CM_4xIO_Link_2[27];
	HwOutputs.ST80_ET200SP_CM_4xIO_Link_2[28] := PlcOutputs.ST80_ET200SP_CM_4xIO_Link_2[28];
	HwOutputs.ST80_ET200SP_CM_4xIO_Link_2[29] := PlcOutputs.ST80_ET200SP_CM_4xIO_Link_2[29];
	HwOutputs.ST80_ET200SP_CM_4xIO_Link_2[30] := PlcOutputs.ST80_ET200SP_CM_4xIO_Link_2[30];
	HwOutputs.ST80_ET200SP_CM_4xIO_Link_2[31] := PlcOutputs.ST80_ET200SP_CM_4xIO_Link_2[31];
	HwOutputs.ST80_ET200SP_CM_4xIO_Link_3[0] := PlcOutputs.ST80_ET200SP_CM_4xIO_Link_3[0];
	HwOutputs.ST80_ET200SP_CM_4xIO_Link_3[1] := PlcOutputs.ST80_ET200SP_CM_4xIO_Link_3[1];
	HwOutputs.ST80_ET200SP_CM_4xIO_Link_3[2] := PlcOutputs.ST80_ET200SP_CM_4xIO_Link_3[2];
	HwOutputs.ST80_ET200SP_CM_4xIO_Link_3[3] := PlcOutputs.ST80_ET200SP_CM_4xIO_Link_3[3];
	HwOutputs.ST80_ET200SP_CM_4xIO_Link_3[4] := PlcOutputs.ST80_ET200SP_CM_4xIO_Link_3[4];
	HwOutputs.ST80_ET200SP_CM_4xIO_Link_3[5] := PlcOutputs.ST80_ET200SP_CM_4xIO_Link_3[5];
	HwOutputs.ST80_ET200SP_CM_4xIO_Link_3[6] := PlcOutputs.ST80_ET200SP_CM_4xIO_Link_3[6];
	HwOutputs.ST80_ET200SP_CM_4xIO_Link_3[7] := PlcOutputs.ST80_ET200SP_CM_4xIO_Link_3[7];
	HwOutputs.ST80_ET200SP_CM_4xIO_Link_3[8] := PlcOutputs.ST80_ET200SP_CM_4xIO_Link_3[8];
	HwOutputs.ST80_ET200SP_CM_4xIO_Link_3[9] := PlcOutputs.ST80_ET200SP_CM_4xIO_Link_3[9];
	HwOutputs.ST80_ET200SP_CM_4xIO_Link_3[10] := PlcOutputs.ST80_ET200SP_CM_4xIO_Link_3[10];
	HwOutputs.ST80_ET200SP_CM_4xIO_Link_3[11] := PlcOutputs.ST80_ET200SP_CM_4xIO_Link_3[11];
	HwOutputs.ST80_ET200SP_CM_4xIO_Link_3[12] := PlcOutputs.ST80_ET200SP_CM_4xIO_Link_3[12];
	HwOutputs.ST80_ET200SP_CM_4xIO_Link_3[13] := PlcOutputs.ST80_ET200SP_CM_4xIO_Link_3[13];
	HwOutputs.ST80_ET200SP_CM_4xIO_Link_3[14] := PlcOutputs.ST80_ET200SP_CM_4xIO_Link_3[14];
	HwOutputs.ST80_ET200SP_CM_4xIO_Link_3[15] := PlcOutputs.ST80_ET200SP_CM_4xIO_Link_3[15];
	HwOutputs.ST80_ET200SP_CM_4xIO_Link_3[16] := PlcOutputs.ST80_ET200SP_CM_4xIO_Link_3[16];
	HwOutputs.ST80_ET200SP_CM_4xIO_Link_3[17] := PlcOutputs.ST80_ET200SP_CM_4xIO_Link_3[17];
	HwOutputs.ST80_ET200SP_CM_4xIO_Link_3[18] := PlcOutputs.ST80_ET200SP_CM_4xIO_Link_3[18];
	HwOutputs.ST80_ET200SP_CM_4xIO_Link_3[19] := PlcOutputs.ST80_ET200SP_CM_4xIO_Link_3[19];
	HwOutputs.ST80_ET200SP_CM_4xIO_Link_3[20] := PlcOutputs.ST80_ET200SP_CM_4xIO_Link_3[20];
	HwOutputs.ST80_ET200SP_CM_4xIO_Link_3[21] := PlcOutputs.ST80_ET200SP_CM_4xIO_Link_3[21];
	HwOutputs.ST80_ET200SP_CM_4xIO_Link_3[22] := PlcOutputs.ST80_ET200SP_CM_4xIO_Link_3[22];
	HwOutputs.ST80_ET200SP_CM_4xIO_Link_3[23] := PlcOutputs.ST80_ET200SP_CM_4xIO_Link_3[23];
	HwOutputs.ST80_ET200SP_CM_4xIO_Link_3[24] := PlcOutputs.ST80_ET200SP_CM_4xIO_Link_3[24];
	HwOutputs.ST80_ET200SP_CM_4xIO_Link_3[25] := PlcOutputs.ST80_ET200SP_CM_4xIO_Link_3[25];
	HwOutputs.ST80_ET200SP_CM_4xIO_Link_3[26] := PlcOutputs.ST80_ET200SP_CM_4xIO_Link_3[26];
	HwOutputs.ST80_ET200SP_CM_4xIO_Link_3[27] := PlcOutputs.ST80_ET200SP_CM_4xIO_Link_3[27];
	HwOutputs.ST80_ET200SP_CM_4xIO_Link_3[28] := PlcOutputs.ST80_ET200SP_CM_4xIO_Link_3[28];
	HwOutputs.ST80_ET200SP_CM_4xIO_Link_3[29] := PlcOutputs.ST80_ET200SP_CM_4xIO_Link_3[29];
	HwOutputs.ST80_ET200SP_CM_4xIO_Link_3[30] := PlcOutputs.ST80_ET200SP_CM_4xIO_Link_3[30];
	HwOutputs.ST80_ET200SP_CM_4xIO_Link_3[31] := PlcOutputs.ST80_ET200SP_CM_4xIO_Link_3[31];
	HwOutputs.ST80_ET200SP_DQ_16x24VDC_0_5A_ST_1 := PlcOutputs.ST80_ET200SP_DQ_16x24VDC_0_5A_ST_1;
	HwOutputs.ST80_ET200SP_DQ_16x24VDC_0_5A_ST_2 := PlcOutputs.ST80_ET200SP_DQ_16x24VDC_0_5A_ST_2;
	HwOutputs.ST80_ET200SP_DQ_16x24VDC_0_5A_ST_3 := PlcOutputs.ST80_ET200SP_DQ_16x24VDC_0_5A_ST_3;
END_FUNCTION
